LIN {X 0,Y 220.868,Z 520.969,A -85,B 0,C 180,E1 -20497.552,E2 -20497.552} C_VEL
LIN {X 0,Y 220.987,Z 520.957,A -85,B 0,C 180,E1 -20502.57,E2 -20502.57} C_VEL
LIN {X 0,Y 221.013,Z 520.952,A -85,B 0,C 180,E1 -20507.138,E2 -20507.138} C_VEL
LIN {X 0,Y 221.2,Z 520.932,A -85,B 0,C 180,E1 -20510.859,E2 -20510.859} C_VEL
LIN {X 0,Y 221.129,Z 520.939,A -85,B 0,C 180,E1 -20514.528,E2 -20514.528} C_VEL
LIN {X 0,Y 221.511,Z 520.89,A -85,B 0,C 180,E1 -20518.181,E2 -20518.181} C_VEL
LIN {X 0,Y 221.506,Z 520.891,A -85,B 0,C 180,E1 -20521.818,E2 -20521.818} C_VEL
LIN {X 0,Y 221.24,Z 520.926,A -85,B 0,C 180,E1 -20527.3,E2 -20527.3} C_VEL
LIN {X 0,Y 221.067,Z 520.947,A -85,B 0,C 180,E1 -20530.996,E2 -20530.996} C_VEL
LIN {X 0,Y 220.978,Z 520.958,A -85,B 0,C 180,E1 -20534.74,E2 -20534.74} C_VEL
LIN {X 0,Y 220.899,Z 520.969,A -85,B 0,C 180,E1 -20538.551,E2 -20538.551} C_VEL
LIN {X 0,Y 220.868,Z 520.97,A -85,B 0,C 180,E1 -20542.664,E2 -20542.664} C_VEL
LIN {X 0,Y 220.866,Z 520.973,A -85,B 0,C 180,E1 -20547.005,E2 -20547.005} C_VEL
LIN {X 0,Y 220.818,Z 520.98,A -85,B 0,C 180,E1 -20550.758,E2 -20550.758} C_VEL
LIN {X 0,Y 220.81,Z 520.981,A -85,B 0,C 180,E1 -20554.953,E2 -20554.953} C_VEL
LIN {X 0,Y 220.892,Z 521.149,A -85,B 0,C 180,E1 -20556.482,E2 -20556.482} C_VEL
LIN {X 0,Y 222.343,Z 528.666,A -85,B 0,C 180,E1 -20561.589,E2 -20561.589} C_VEL
LIN {X 0,Y 223.777,Z 535.991,A -85,B 0,C 180,E1 -20566.296,E2 -20566.296} C_VEL
LIN {X 0,Y 225.008,Z 542.365,A -85,B 0,C 180,E1 -20570.186,E2 -20570.186} C_VEL
LIN {X 0,Y 225.036,Z 544.358,A -85,B 0,C 180,E1 -20571.346,E2 -20571.346} C_VEL
LIN {X 0,Y 222.99,Z 553.544,A -85,B 0,C 180,E1 -20576.527,E2 -20576.527} C_VEL
LIN {X 0,Y 221.333,Z 562.382,A -85,B 0,C 180,E1 -20581.395,E2 -20581.395} C_VEL
LIN {X 0,Y 222.533,Z 577.013,A -85,B 0,C 180,E1 -20582.449,E2 -20582.449} C_VEL
LIN {X 0,Y 223.287,Z 589.6,A -85,B 0,C 180,E1 -20583.692,E2 -20583.692} C_VEL
LIN {X 0,Y 223.376,Z 591.056,A -85,B 0,C 180,E1 -20583.862,E2 -20583.862} C_VEL
LIN {X 0,Y 222.993,Z 596.491,A -85,B 0,C 180,E1 -20584.484,E2 -20584.484} C_VEL
LIN {X 0,Y 220.374,Z 605.07,A -85,B 0,C 180,E1 -20585.546,E2 -20585.546} C_VEL
LIN {X 0,Y 217.508,Z 613.354,A -85,B 0,C 180,E1 -20586.792,E2 -20586.792} C_VEL
LIN {X 0,Y 216.761,Z 618.17,A -85,B 0,C 180,E1 -20587.69,E2 -20587.69} C_VEL
LIN {X 0,Y 216.495,Z 628.791,A -85,B 0,C 180,E1 -20590.028,E2 -20590.028} C_VEL
LIN {X 0,Y 215.182,Z 637.685,A -85,B 0,C 180,E1 -20592.416,E2 -20592.416} C_VEL
LIN {X 0,Y 213.795,Z 646.126,A -85,B 0,C 180,E1 -20595.241,E2 -20595.241} C_VEL
LIN {X 0,Y 213.228,Z 652.944,A -85,B 0,C 180,E1 -20598.112,E2 -20598.112} C_VEL
LIN {X 0,Y 213.044,Z 659.023,A -85,B 0,C 180,E1 -20601.395,E2 -20601.395} C_VEL
LIN {X 0,Y 213.394,Z 663.111,A -85,B 0,C 180,E1 -20604.33,E2 -20604.33} C_VEL
LIN {X 0,Y 213.6,Z 665.077,A -85,B 0,C 180,E1 -20606.227,E2 -20606.227} C_VEL
LIN {X 0,Y 213.964,Z 666.582,A -85,B 0,C 180,E1 -20608.118,E2 -20608.118} C_VEL
LIN {X 0,Y 214.253,Z 667.619,A -85,B 0,C 180,E1 -20610,E2 -20610} C_VEL
LIN {X 0,Y 213.722,Z 668.07,A -85,B 0,C 180,E1 -20611.885,E2 -20611.885} C_VEL
LIN {X 0,Y 213.262,Z 668.071,A -85,B 0,C 180,E1 -20613.779,E2 -20613.779} C_VEL
LIN {X 0,Y 212.95,Z 667.676,A -85,B 0,C 180,E1 -20615.682,E2 -20615.682} C_VEL
LIN {X 0,Y 212.44,Z 665.683,A -85,B 0,C 180,E1 -20619.521,E2 -20619.521} C_VEL
LIN {X 0,Y 212.569,Z 664.115,A -85,B 0,C 180,E1 -20621.442,E2 -20621.442} C_VEL
LIN {X 0,Y 213.6,Z 659.748,A -85,B 0,C 180,E1 -20625.262,E2 -20625.262} C_VEL
LIN {X 0,Y 214.967,Z 655.403,A -85,B 0,C 180,E1 -20628.095,E2 -20628.095} C_VEL
LIN {X 0,Y 217.648,Z 649.066,A -85,B 0,C 180,E1 -20631.302,E2 -20631.302} C_VEL
LIN {X 0,Y 221.044,Z 641.112,A -85,B 0,C 180,E1 -20634.415,E2 -20634.415} C_VEL
LIN {X 0,Y 224.313,Z 631.288,A -85,B 0,C 180,E1 -20637.525,E2 -20637.525} C_VEL
LIN {X 0,Y 227.265,Z 621.289,A -85,B 0,C 180,E1 -20640.116,E2 -20640.116} C_VEL
LIN {X 0,Y 229.051,Z 612.146,A -85,B 0,C 180,E1 -20642.217,E2 -20642.217} C_VEL
LIN {X 0,Y 230.395,Z 601.122,A -85,B 0,C 180,E1 -20644.552,E2 -20644.552} C_VEL
LIN {X 0,Y 230.791,Z 590.585,A -85,B 0,C 180,E1 -20646.665,E2 -20646.665} C_VEL
LIN {X 0,Y 230.404,Z 579.42,A -85,B 0,C 180,E1 -20648.907,E2 -20648.907} C_VEL
LIN {X 0,Y 229.373,Z 570.02,A -85,B 0,C 180,E1 -20650.835,E2 -20650.835} C_VEL
LIN {X 0,Y 228.281,Z 563.015,A -85,B 0,C 180,E1 -20652.364,E2 -20652.364} C_VEL
LIN {X 0,Y 225.952,Z 556.827,A -85,B 0,C 180,E1 -20654.258,E2 -20654.258} C_VEL
LIN {X 0,Y 223.212,Z 551.163,A -85,B 0,C 180,E1 -20656.437,E2 -20656.437} C_VEL
LIN {X 0,Y 222.42,Z 548.881,A -85,B 0,C 180,E1 -20657.206,E2 -20657.206} C_VEL
LIN {X 0,Y 218.789,Z 542.503,A -85,B 0,C 180,E1 -20660.551,E2 -20660.551} C_VEL
LIN {X 0,Y 217.55,Z 538.888,A -85,B 0,C 180,E1 -20662.279,E2 -20662.279} C_VEL
LIN {X 0,Y 217.174,Z 536.934,A -85,B 0,C 180,E1 -20664.374,E2 -20664.374} C_VEL
LIN {X 0,Y 216.367,Z 533.433,A -85,B 0,C 180,E1 -20668.688,E2 -20668.688} C_VEL
LIN {X 0,Y 215.819,Z 530.571,A -85,B 0,C 180,E1 -20672.878,E2 -20672.878} C_VEL
LIN {X 0,Y 215.351,Z 528.348,A -85,B 0,C 180,E1 -20676.945,E2 -20676.945} C_VEL
LIN {X 0,Y 215.107,Z 527.422,A -85,B 0,C 180,E1 -20679.213,E2 -20679.213} C_VEL
LIN {X 0,Y 216.79,Z 529.004,A -85,B 0,C 180,E1 -20682.175,E2 -20682.175} C_VEL
LIN {X 0,Y 219.429,Z 530.078,A -85,B 0,C 180,E1 -20685.154,E2 -20685.154} C_VEL
LIN {X 0,Y 220.989,Z 532.089,A -85,B 0,C 180,E1 -20686.904,E2 -20686.904} C_VEL
LIN {X 0,Y 222.543,Z 533.032,A -85,B 0,C 180,E1 -20688.238,E2 -20688.238} C_VEL
LIN {X 0,Y 224.34,Z 536.433,A -85,B 0,C 180,E1 -20690.145,E2 -20690.145} C_VEL
LIN {X 0,Y 225.36,Z 537.698,A -85,B 0,C 180,E1 -20691.03,E2 -20691.03} C_VEL
LIN {X 0,Y 230.369,Z 546.87,A -85,B 0,C 180,E1 -20695.625,E2 -20695.625} C_VEL
LIN {X 0,Y 232.402,Z 551.236,A -85,B 0,C 180,E1 -20697.547,E2 -20697.547} C_VEL
LIN {X 0,Y 235.12,Z 559.958,A -85,B 0,C 180,E1 -20700.857,E2 -20700.857} C_VEL
LIN {X 0,Y 236.611,Z 566.893,A -85,B 0,C 180,E1 -20703.406,E2 -20703.406} C_VEL
LIN {X 0,Y 237.291,Z 573.898,A -85,B 0,C 180,E1 -20705.951,E2 -20705.951} C_VEL
LIN {X 0,Y 233.871,Z 582.058,A -85,B 0,C 180,E1 -20708.135,E2 -20708.135} C_VEL
LIN {X 0,Y 230.347,Z 589.283,A -85,B 0,C 180,E1 -20710.549,E2 -20710.549} C_VEL
LIN {X 0,Y 226.712,Z 595.941,A -85,B 0,C 180,E1 -20713.445,E2 -20713.445} C_VEL
LIN {X 0,Y 223.496,Z 601.099,A -85,B 0,C 180,E1 -20716.441,E2 -20716.441} C_VEL
LIN {X 0,Y 220.741,Z 604.875,A -85,B 0,C 180,E1 -20719.531,E2 -20719.531} C_VEL
LIN {X 0,Y 218.492,Z 607.379,A -85,B 0,C 180,E1 -20722.706,E2 -20722.706} C_VEL
LIN {X 0,Y 217.166,Z 608.443,A -85,B 0,C 180,E1 -20725.021,E2 -20725.021} C_VEL
LIN {X 0,Y 215.688,Z 608.843,A -85,B 0,C 180,E1 -20728.384,E2 -20728.384} C_VEL
LIN {X 0,Y 214.787,Z 608.01,A -85,B 0,C 180,E1 -20731.707,E2 -20731.707} C_VEL
LIN {X 0,Y 214.36,Z 606.025,A -85,B 0,C 180,E1 -20734.95,E2 -20734.95} C_VEL
LIN {X 0,Y 214.38,Z 602.431,A -85,B 0,C 180,E1 -20738.527,E2 -20738.527} C_VEL
LIN {X 0,Y 214.977,Z 597.143,A -85,B 0,C 180,E1 -20742.145,E2 -20742.145} C_VEL
LIN {X 0,Y 215.807,Z 591.954,A -85,B 0,C 180,E1 -20744.852,E2 -20744.852} C_VEL
LIN {X 0,Y 216.835,Z 585.672,A -85,B 0,C 180,E1 -20747.512,E2 -20747.512} C_VEL
LIN {X 0,Y 218.123,Z 578.071,A -85,B 0,C 180,E1 -20750.135,E2 -20750.135} C_VEL
LIN {X 0,Y 219.642,Z 569.436,A -85,B 0,C 180,E1 -20752.558,E2 -20752.558} C_VEL
LIN {X 0,Y 221.381,Z 558.618,A -85,B 0,C 180,E1 -20755.028,E2 -20755.028} C_VEL
LIN {X 0,Y 222.361,Z 551.653,A -85,B 0,C 180,E1 -20756.349,E2 -20756.349} C_VEL
LIN {X 0,Y 219.673,Z 541.039,A -85,B 0,C 180,E1 -20758.406,E2 -20758.406} C_VEL
LIN {X 0,Y 216.303,Z 529.758,A -85,B 0,C 180,E1 -20760.297,E2 -20760.297} C_VEL
LIN {X 0,Y 213.826,Z 521.856,A -85,B 0,C 180,E1 -20761.471,E2 -20761.471} C_VEL
LIN {X 0,Y 213.803,Z 521.854,A -85,B 0,C 180,E1 -20764.701,E2 -20764.701} C_VEL
LIN {X 0,Y 213.802,Z 521.852,A -85,B 0,C 180,E1 -20768.802,E2 -20768.802} C_VEL
LIN {X 0,Y 213.926,Z 521.838,A -85,B 0,C 180,E1 -20772.802,E2 -20772.802} C_VEL
LIN {X 0,Y 213.948,Z 521.835,A -85,B 0,C 180,E1 -20776.706,E2 -20776.706} C_VEL
LIN {X 0,Y 214.14,Z 521.81,A -85,B 0,C 180,E1 -20780.555,E2 -20780.555} C_VEL
LIN {X 0,Y 214.093,Z 521.815,A -85,B 0,C 180,E1 -20784.348,E2 -20784.348} C_VEL
LIN {X 0,Y 214.447,Z 521.77,A -85,B 0,C 180,E1 -20788.122,E2 -20788.122} C_VEL
LIN {X 0,Y 214.54,Z 521.759,A -85,B 0,C 180,E1 -20790,E2 -20790} C_VEL
LIN {X 0,Y 214.446,Z 521.771,A -85,B 0,C 180,E1 -20791.878,E2 -20791.878} C_VEL
LIN {X 0,Y 214.185,Z 521.802,A -85,B 0,C 180,E1 -20797.542,E2 -20797.542} C_VEL
LIN {X 0,Y 213.998,Z 521.83,A -85,B 0,C 180,E1 -20801.364,E2 -20801.364} C_VEL
LIN {X 0,Y 213.921,Z 521.838,A -85,B 0,C 180,E1 -20805.238,E2 -20805.238} C_VEL
LIN {X 0,Y 213.838,Z 521.848,A -85,B 0,C 180,E1 -20809.187,E2 -20809.187} C_VEL
LIN {X 0,Y 213.808,Z 521.852,A -85,B 0,C 180,E1 -20813.231,E2 -20813.231} C_VEL
LIN {X 0,Y 213.792,Z 521.854,A -85,B 0,C 180,E1 -20817.428,E2 -20817.428} C_VEL
LIN {X 0,Y 213.761,Z 521.856,A -85,B 0,C 180,E1 -20821.738,E2 -20821.738} C_VEL
LIN {X 0,Y 213.746,Z 521.857,A -85,B 0,C 180,E1 -20826.288,E2 -20826.288} C_VEL
LIN {X 0,Y 213.705,Z 521.864,A -85,B 0,C 180,E1 -20831.127,E2 -20831.127} C_VEL
LIN {X 0,Y 213.705,Z 521.862,A -85,B 0,C 180,E1 -20833.679,E2 -20833.679} C_VEL
LIN {X 0,Y 213.705,Z 521.863,A -85,B 0,C 180,E1 -20836.344,E2 -20836.344} C_VEL
LIN {X 0,Y 213.719,Z 521.863,A -85,B 0,C 180,E1 -20839.143,E2 -20839.143} C_VEL
LIN {X 0,Y 213.746,Z 521.858,A -85,B 0,C 180,E1 -20843.711,E2 -20843.711} C_VEL
LIN {X 0,Y 213.797,Z 521.852,A -85,B 0,C 180,E1 -20848.724,E2 -20848.724} C_VEL
LIN {X 0,Y 213.828,Z 521.848,A -85,B 0,C 180,E1 -20852.603,E2 -20852.603} C_VEL
LIN {X 0,Y 213.821,Z 521.85,A -85,B 0,C 180,E1 -20856.973,E2 -20856.973} C_VEL
LIN {X 0,Y 213.946,Z 521.836,A -85,B 0,C 180,E1 -20862.803,E2 -20862.803} C_VEL
LIN {X 0,Y 213.955,Z 521.832,A -85,B 0,C 180,E1 -20866.706,E2 -20866.706} C_VEL
LIN {X 0,Y 214.138,Z 521.81,A -85,B 0,C 180,E1 -20870.555,E2 -20870.555} C_VEL
LIN {X 0,Y 214.09,Z 521.815,A -85,B 0,C 180,E1 -20874.348,E2 -20874.348} C_VEL
LIN {X 0,Y 214.444,Z 521.77,A -85,B 0,C 180,E1 -20878.121,E2 -20878.121} C_VEL
LIN {X 0,Y 214.543,Z 521.759,A -85,B 0,C 180,E1 -20880,E2 -20880} C_VEL
LIN {X 0,Y 214.439,Z 521.771,A -85,B 0,C 180,E1 -20881.878,E2 -20881.878} C_VEL
LIN {X 0,Y 214.182,Z 521.804,A -85,B 0,C 180,E1 -20887.542,E2 -20887.542} C_VEL
LIN {X 0,Y 213.998,Z 521.825,A -85,B 0,C 180,E1 -20891.364,E2 -20891.364} C_VEL
LIN {X 0,Y 213.914,Z 521.838,A -85,B 0,C 180,E1 -20895.238,E2 -20895.238} C_VEL
LIN {X 0,Y 213.82,Z 521.849,A -85,B 0,C 180,E1 -20899.189,E2 -20899.189} C_VEL
LIN {X 0,Y 213.803,Z 521.851,A -85,B 0,C 180,E1 -20903.232,E2 -20903.232} C_VEL
LIN {X 0,Y 213.787,Z 521.853,A -85,B 0,C 180,E1 -20907.428,E2 -20907.428} C_VEL
LIN {X 0,Y 213.759,Z 521.861,A -85,B 0,C 180,E1 -20911.739,E2 -20911.739} C_VEL
LIN {X 0,Y 213.83,Z 522.009,A -85,B 0,C 180,E1 -20916.053,E2 -20916.053} C_VEL
LIN {X 0,Y 215.117,Z 528.734,A -85,B 0,C 180,E1 -20920.799,E2 -20920.799} C_VEL
LIN {X 0,Y 216.124,Z 533.968,A -85,B 0,C 180,E1 -20924.324,E2 -20924.324} C_VEL
LIN {X 0,Y 217.586,Z 541.147,A -85,B 0,C 180,E1 -20928.934,E2 -20928.934} C_VEL
LIN {X 0,Y 217.963,Z 544.027,A -85,B 0,C 180,E1 -20930.701,E2 -20930.701} C_VEL
LIN {X 0,Y 217.58,Z 546.471,A -85,B 0,C 180,E1 -20932.141,E2 -20932.141} C_VEL
LIN {X 0,Y 215.903,Z 553.764,A -85,B 0,C 180,E1 -20936.401,E2 -20936.401} C_VEL
LIN {X 0,Y 214.425,Z 561.289,A -85,B 0,C 180,E1 -20940.752,E2 -20940.752} C_VEL
LIN {X 0,Y 215.6,Z 576.166,A -85,B 0,C 180,E1 -20941.87,E2 -20941.87} C_VEL
LIN {X 0,Y 216.289,Z 589.084,A -85,B 0,C 180,E1 -20943.202,E2 -20943.202} C_VEL
LIN {X 0,Y 216.665,Z 601.267,A -85,B 0,C 180,E1 -20944.803,E2 -20944.803} C_VEL
LIN {X 0,Y 216.83,Z 612.403,A -85,B 0,C 180,E1 -20946.606,E2 -20946.606} C_VEL
LIN {X 0,Y 216.761,Z 618.17,A -85,B 0,C 180,E1 -20947.69,E2 -20947.69} C_VEL
LIN {X 0,Y 215.93,Z 622.846,A -85,B 0,C 180,E1 -20948.642,E2 -20948.642} C_VEL
LIN {X 0,Y 214.068,Z 627.214,A -85,B 0,C 180,E1 -20949.61,E2 -20949.61} C_VEL
LIN {X 0,Y 209.48,Z 635.189,A -85,B 0,C 180,E1 -20951.703,E2 -20951.703} C_VEL
LIN {X 0,Y 207.845,Z 638.989,A -85,B 0,C 180,E1 -20952.892,E2 -20952.892} C_VEL
LIN {X 0,Y 207.543,Z 640.232,A -85,B 0,C 180,E1 -20953.312,E2 -20953.312} C_VEL
LIN {X 0,Y 206.563,Z 647.939,A -85,B 0,C 180,E1 -20956.222,E2 -20956.222} C_VEL
LIN {X 0,Y 206.06,Z 654.149,A -85,B 0,C 180,E1 -20959.188,E2 -20959.188} C_VEL
LIN {X 0,Y 206.046,Z 659.04,A -85,B 0,C 180,E1 -20962.159,E2 -20962.159} C_VEL
LIN {X 0,Y 206.462,Z 662.744,A -85,B 0,C 180,E1 -20965.118,E2 -20965.118} C_VEL
LIN {X 0,Y 206.931,Z 665.294,A -85,B 0,C 180,E1 -20968.054,E2 -20968.054} C_VEL
LIN {X 0,Y 207.253,Z 666.387,A -85,B 0,C 180,E1 -20970,E2 -20970} C_VEL
LIN {X 0,Y 206.697,Z 666.887,A -85,B 0,C 180,E1 -20971.949,E2 -20971.949} C_VEL
LIN {X 0,Y 206.201,Z 666.971,A -85,B 0,C 180,E1 -20973.909,E2 -20973.909} C_VEL
LIN {X 0,Y 205.879,Z 666.632,A -85,B 0,C 180,E1 -20975.878,E2 -20975.878} C_VEL
LIN {X 0,Y 205.38,Z 664.743,A -85,B 0,C 180,E1 -20979.852,E2 -20979.852} C_VEL
LIN {X 0,Y 205.954,Z 661.373,A -85,B 0,C 180,E1 -20983.82,E2 -20983.82} C_VEL
LIN {X 0,Y 207.628,Z 656.377,A -85,B 0,C 180,E1 -20987.737,E2 -20987.737} C_VEL
LIN {X 0,Y 209.681,Z 651.515,A -85,B 0,C 180,E1 -20990.606,E2 -20990.606} C_VEL
LIN {X 0,Y 212.984,Z 644.514,A -85,B 0,C 180,E1 -20993.843,E2 -20993.843} C_VEL
LIN {X 0,Y 215.983,Z 637.184,A -85,B 0,C 180,E1 -20996.579,E2 -20996.579} C_VEL
LIN {X 0,Y 219.013,Z 628.599,A -85,B 0,C 180,E1 -20999.234,E2 -20999.234} C_VEL
LIN {X 0,Y 222.103,Z 617.956,A -85,B 0,C 180,E1 -21002.007,E2 -21002.007} C_VEL
LIN {X 0,Y 224.097,Z 606.805,A -85,B 0,C 180,E1 -21004.631,E2 -21004.631} C_VEL
LIN {X 0,Y 225.205,Z 596.058,A -85,B 0,C 180,E1 -21006.971,E2 -21006.971} C_VEL
LIN {X 0,Y 225.365,Z 583.627,A -85,B 0,C 180,E1 -21009.637,E2 -21009.637} C_VEL
LIN {X 0,Y 224.586,Z 571.366,A -85,B 0,C 180,E1 -21012.343,E2 -21012.343} C_VEL
LIN {X 0,Y 224.02,Z 567.653,A -85,B 0,C 180,E1 -21013.235,E2 -21013.235} C_VEL
LIN {X 0,Y 222.549,Z 562.746,A -85,B 0,C 180,E1 -21014.783,E2 -21014.783} C_VEL
LIN {X 0,Y 219.891,Z 556.62,A -85,B 0,C 180,E1 -21017.241,E2 -21017.241} C_VEL
LIN {X 0,Y 219.193,Z 554.511,A -85,B 0,C 180,E1 -21018.048,E2 -21018.048} C_VEL
LIN {X 0,Y 215.995,Z 547.879,A -85,B 0,C 180,E1 -21021.591,E2 -21021.591} C_VEL
LIN {X 0,Y 215.084,Z 545.09,A -85,B 0,C 180,E1 -21022.995,E2 -21022.995} C_VEL
LIN {X 0,Y 212.196,Z 539.413,A -85,B 0,C 180,E1 -21028.419,E2 -21028.419} C_VEL
LIN {X 0,Y 211.575,Z 536.634,A -85,B 0,C 180,E1 -21032.287,E2 -21032.287} C_VEL
LIN {X 0,Y 212.378,Z 534.76,A -85,B 0,C 180,E1 -21037.119,E2 -21037.119} C_VEL
LIN {X 0,Y 213.373,Z 534.411,A -85,B 0,C 180,E1 -21039.263,E2 -21039.263} C_VEL
LIN {X 0,Y 215.359,Z 536.111,A -85,B 0,C 180,E1 -21042.921,E2 -21042.921} C_VEL
LIN {X 0,Y 217.092,Z 536.896,A -85,B 0,C 180,E1 -21044.99,E2 -21044.99} C_VEL
LIN {X 0,Y 218.737,Z 538.899,A -85,B 0,C 180,E1 -21047.003,E2 -21047.003} C_VEL
LIN {X 0,Y 219.815,Z 539.821,A -85,B 0,C 180,E1 -21048.09,E2 -21048.09} C_VEL
LIN {X 0,Y 222.545,Z 545.038,A -85,B 0,C 180,E1 -21051.307,E2 -21051.307} C_VEL
LIN {X 0,Y 226.246,Z 552.522,A -85,B 0,C 180,E1 -21055.301,E2 -21055.301} C_VEL
LIN {X 0,Y 227.969,Z 556.735,A -85,B 0,C 180,E1 -21057.254,E2 -21057.254} C_VEL
LIN {X 0,Y 230.367,Z 566.269,A -85,B 0,C 180,E1 -21061.131,E2 -21061.131} C_VEL
LIN {X 0,Y 231.268,Z 573.398,A -85,B 0,C 180,E1 -21063.921,E2 -21063.921} C_VEL
LIN {X 0,Y 231.367,Z 576.788,A -85,B 0,C 180,E1 -21065.229,E2 -21065.229} C_VEL
LIN {X 0,Y 227.544,Z 584.936,A -85,B 0,C 180,E1 -21067.557,E2 -21067.557} C_VEL
LIN {X 0,Y 223.344,Z 592.775,A -85,B 0,C 180,E1 -21070.425,E2 -21070.425} C_VEL
LIN {X 0,Y 220.216,Z 598.009,A -85,B 0,C 180,E1 -21072.909,E2 -21072.909} C_VEL
LIN {X 0,Y 216.841,Z 602.912,A -85,B 0,C 180,E1 -21075.992,E2 -21075.992} C_VEL
LIN {X 0,Y 213.967,Z 606.475,A -85,B 0,C 180,E1 -21079.176,E2 -21079.176} C_VEL
LIN {X 0,Y 211.991,Z 608.442,A -85,B 0,C 180,E1 -21081.833,E2 -21081.833} C_VEL
LIN {X 0,Y 209.967,Z 609.808,A -85,B 0,C 180,E1 -21085.344,E2 -21085.344} C_VEL
LIN {X 0,Y 208.5,Z 609.88,A -85,B 0,C 180,E1 -21088.789,E2 -21088.789} C_VEL
LIN {X 0,Y 207.648,Z 608.693,A -85,B 0,C 180,E1 -21092.204,E2 -21092.204} C_VEL
LIN {X 0,Y 207.279,Z 606.371,A -85,B 0,C 180,E1 -21095.536,E2 -21095.536} C_VEL
LIN {X 0,Y 207.353,Z 602.965,A -85,B 0,C 180,E1 -21098.779,E2 -21098.779} C_VEL
LIN {X 0,Y 207.858,Z 598.439,A -85,B 0,C 180,E1 -21101.939,E2 -21101.939} C_VEL
LIN {X 0,Y 208.787,Z 592.729,A -85,B 0,C 180,E1 -21105.017,E2 -21105.017} C_VEL
LIN {X 0,Y 209.913,Z 585.863,A -85,B 0,C 180,E1 -21107.962,E2 -21107.962} C_VEL
LIN {X 0,Y 211.369,Z 577.551,A -85,B 0,C 180,E1 -21110.82,E2 -21110.82} C_VEL
LIN {X 0,Y 213.189,Z 567.487,A -85,B 0,C 180,E1 -21113.602,E2 -21113.602} C_VEL
LIN {X 0,Y 214.866,Z 557.035,A -85,B 0,C 180,E1 -21115.911,E2 -21115.911} C_VEL
LIN {X 0,Y 215.445,Z 553.444,A -85,B 0,C 180,E1 -21116.6,E2 -21116.6} C_VEL
LIN {X 0,Y 213.299,Z 544.314,A -85,B 0,C 180,E1 -21118.461,E2 -21118.461} C_VEL
LIN {X 0,Y 209.808,Z 532.392,A -85,B 0,C 180,E1 -21120.593,E2 -21120.593} C_VEL
LIN {X 0,Y 206.77,Z 522.733,A -85,B 0,C 180,E1 -21122.097,E2 -21122.097} C_VEL
LIN {X 0,Y 206.758,Z 522.73,A -85,B 0,C 180,E1 -21126.604,E2 -21126.604} C_VEL
LIN {X 0,Y 206.872,Z 522.716,A -85,B 0,C 180,E1 -21132.196,E2 -21132.196} C_VEL
LIN {X 0,Y 206.889,Z 522.714,A -85,B 0,C 180,E1 -21136.244,E2 -21136.244} C_VEL
LIN {X 0,Y 207.084,Z 522.689,A -85,B 0,C 180,E1 -21140.23,E2 -21140.23} C_VEL
LIN {X 0,Y 207.055,Z 522.692,A -85,B 0,C 180,E1 -21144.155,E2 -21144.155} C_VEL
LIN {X 0,Y 207.384,Z 522.65,A -85,B 0,C 180,E1 -21148.058,E2 -21148.058} C_VEL
LIN {X 0,Y 207.507,Z 522.636,A -85,B 0,C 180,E1 -21150,E2 -21150} C_VEL
LIN {X 0,Y 207.382,Z 522.65,A -85,B 0,C 180,E1 -21151.942,E2 -21151.942} C_VEL
LIN {X 0,Y 207.13,Z 522.68,A -85,B 0,C 180,E1 -21157.8,E2 -21157.8} C_VEL
LIN {X 0,Y 206.921,Z 522.709,A -85,B 0,C 180,E1 -21161.758,E2 -21161.758} C_VEL
LIN {X 0,Y 206.857,Z 522.715,A -85,B 0,C 180,E1 -21165.771,E2 -21165.771} C_VEL
LIN {X 0,Y 206.766,Z 522.727,A -85,B 0,C 180,E1 -21169.871,E2 -21169.871} C_VEL
LIN {X 0,Y 206.743,Z 522.729,A -85,B 0,C 180,E1 -21174.074,E2 -21174.074} C_VEL
LIN {X 0,Y 206.693,Z 522.736,A -85,B 0,C 180,E1 -21178.426,E2 -21178.426} C_VEL
LIN {X 0,Y 206.698,Z 522.738,A -85,B 0,C 180,E1 -21182.958,E2 -21182.958} C_VEL
LIN {X 0,Y 206.676,Z 522.739,A -85,B 0,C 180,E1 -21187.741,E2 -21187.741} C_VEL
LIN {X 0,Y 206.637,Z 522.742,A -85,B 0,C 180,E1 -21191.56,E2 -21191.56} C_VEL
LIN {X 0,Y 206.633,Z 522.745,A -85,B 0,C 180,E1 -21195.582,E2 -21195.582} C_VEL
LIN {X 0,Y 206.662,Z 522.739,A -85,B 0,C 180,E1 -21199.748,E2 -21199.748} C_VEL
LIN {X 0,Y 206.701,Z 522.736,A -85,B 0,C 180,E1 -21204.688,E2 -21204.688} C_VEL
LIN {X 0,Y 206.725,Z 522.73,A -85,B 0,C 180,E1 -21209.339,E2 -21209.339} C_VEL
LIN {X 0,Y 206.733,Z 522.732,A -85,B 0,C 180,E1 -21213.771,E2 -21213.771} C_VEL
LIN {X 0,Y 206.741,Z 522.728,A -85,B 0,C 180,E1 -21218.041,E2 -21218.041} C_VEL
LIN {X 0,Y 206.875,Z 522.714,A -85,B 0,C 180,E1 -21222.196,E2 -21222.196} C_VEL
LIN {X 0,Y 206.898,Z 522.709,A -85,B 0,C 180,E1 -21226.244,E2 -21226.244} C_VEL
LIN {X 0,Y 207.081,Z 522.688,A -85,B 0,C 180,E1 -21230.23,E2 -21230.23} C_VEL
LIN {X 0,Y 207.052,Z 522.691,A -85,B 0,C 180,E1 -21234.155,E2 -21234.155} C_VEL
LIN {X 0,Y 207.38,Z 522.65,A -85,B 0,C 180,E1 -21238.057,E2 -21238.057} C_VEL
LIN {X 0,Y 207.509,Z 522.635,A -85,B 0,C 180,E1 -21239.999,E2 -21239.999} C_VEL
LIN {X 0,Y 207.375,Z 522.651,A -85,B 0,C 180,E1 -21241.942,E2 -21241.942} C_VEL
LIN {X 0,Y 207.127,Z 522.682,A -85,B 0,C 180,E1 -21247.8,E2 -21247.8} C_VEL
LIN {X 0,Y 206.922,Z 522.706,A -85,B 0,C 180,E1 -21251.758,E2 -21251.758} C_VEL
LIN {X 0,Y 206.847,Z 522.717,A -85,B 0,C 180,E1 -21255.772,E2 -21255.772} C_VEL
LIN {X 0,Y 206.857,Z 522.716,A -85,B 0,C 180,E1 -21257.954,E2 -21257.954} C_VEL
LIN {X 0,Y 206.746,Z 522.73,A -85,B 0,C 180,E1 -21263.39,E2 -21263.39} C_VEL
LIN {X 0,Y 206.689,Z 522.738,A -85,B 0,C 180,E1 -21268.427,E2 -21268.427} C_VEL
LIN {X 0,Y 206.697,Z 522.741,A -85,B 0,C 180,E1 -21272.958,E2 -21272.958} C_VEL
LIN {X 0,Y 206.778,Z 522.885,A -85,B 0,C 180,E1 -21275.646,E2 -21275.646} C_VEL
LIN {X 0,Y 207.894,Z 528.772,A -85,B 0,C 180,E1 -21279.964,E2 -21279.964} C_VEL
LIN {X 0,Y 208.919,Z 533.975,A -85,B 0,C 180,E1 -21283.599,E2 -21283.599} C_VEL
LIN {X 0,Y 210.272,Z 540.642,A -85,B 0,C 180,E1 -21288.051,E2 -21288.051} C_VEL
LIN {X 0,Y 210.883,Z 544.806,A -85,B 0,C 180,E1 -21290.713,E2 -21290.713} C_VEL
LIN {X 0,Y 209.874,Z 549.36,A -85,B 0,C 180,E1 -21293.483,E2 -21293.483} C_VEL
LIN {X 0,Y 208.365,Z 555.987,A -85,B 0,C 180,E1 -21297.482,E2 -21297.482} C_VEL
LIN {X 0,Y 207.508,Z 560.273,A -85,B 0,C 180,E1 -21300.065,E2 -21300.065} C_VEL
LIN {X 0,Y 208.674,Z 575.929,A -85,B 0,C 180,E1 -21301.304,E2 -21301.304} C_VEL
LIN {X 0,Y 209.337,Z 589.369,A -85,B 0,C 180,E1 -21302.779,E2 -21302.779} C_VEL
LIN {X 0,Y 209.668,Z 601.548,A -85,B 0,C 180,E1 -21304.473,E2 -21304.473} C_VEL
LIN {X 0,Y 209.784,Z 613.555,A -85,B 0,C 180,E1 -21306.558,E2 -21306.558} C_VEL
LIN {X 0,Y 209.567,Z 624.575,A -85,B 0,C 180,E1 -21308.907,E2 -21308.907} C_VEL
LIN {X 0,Y 209.255,Z 630.454,A -85,B 0,C 180,E1 -21310.375,E2 -21310.375} C_VEL
LIN {X 0,Y 207.847,Z 638.667,A -85,B 0,C 180,E1 -21312.791,E2 -21312.791} C_VEL
LIN {X 0,Y 207.543,Z 640.232,A -85,B 0,C 180,E1 -21313.312,E2 -21313.312} C_VEL
LIN {X 0,Y 206.299,Z 643.767,A -85,B 0,C 180,E1 -21314.585,E2 -21314.585} C_VEL
LIN {X 0,Y 202.81,Z 648.792,A -85,B 0,C 180,E1 -21316.778,E2 -21316.778} C_VEL
LIN {X 0,Y 199.677,Z 653.18,A -85,B 0,C 180,E1 -21319.157,E2 -21319.157} C_VEL
LIN {X 0,Y 198.997,Z 655.644,A -85,B 0,C 180,E1 -21320.684,E2 -21320.684} C_VEL
LIN {X 0,Y 199.29,Z 660.154,A -85,B 0,C 180,E1 -21323.927,E2 -21323.927} C_VEL
LIN {X 0,Y 199.535,Z 662.306,A -85,B 0,C 180,E1 -21325.961,E2 -21325.961} C_VEL
LIN {X 0,Y 199.897,Z 663.978,A -85,B 0,C 180,E1 -21327.985,E2 -21327.985} C_VEL
LIN {X 0,Y 200.248,Z 665.132,A -85,B 0,C 180,E1 -21330,E2 -21330} C_VEL
LIN {X 0,Y 199.667,Z 665.683,A -85,B 0,C 180,E1 -21332.017,E2 -21332.017} C_VEL
LIN {X 0,Y 198.787,Z 665.575,A -85,B 0,C 180,E1 -21336.089,E2 -21336.089} C_VEL
LIN {X 0,Y 198.347,Z 663.816,A -85,B 0,C 180,E1 -21340.205,E2 -21340.205} C_VEL
LIN {X 0,Y 199.001,Z 660.586,A -85,B 0,C 180,E1 -21344.313,E2 -21344.313} C_VEL
LIN {X 0,Y 200.247,Z 657.129,A -85,B 0,C 180,E1 -21347.357,E2 -21347.357} C_VEL
LIN {X 0,Y 202.138,Z 652.758,A -85,B 0,C 180,E1 -21350.346,E2 -21350.346} C_VEL
LIN {X 0,Y 205.4,Z 646.414,A -85,B 0,C 180,E1 -21353.706,E2 -21353.706} C_VEL
LIN {X 0,Y 208.592,Z 639.711,A -85,B 0,C 180,E1 -21356.515,E2 -21356.515} C_VEL
LIN {X 0,Y 212.302,Z 630.231,A -85,B 0,C 180,E1 -21359.773,E2 -21359.773} C_VEL
LIN {X 0,Y 215.602,Z 620.479,A -85,B 0,C 180,E1 -21362.538,E2 -21362.538} C_VEL
LIN {X 0,Y 218.153,Z 609.035,A -85,B 0,C 180,E1 -21365.443,E2 -21365.443} C_VEL
LIN {X 0,Y 219.586,Z 598.979,A -85,B 0,C 180,E1 -21367.805,E2 -21367.805} C_VEL
LIN {X 0,Y 220.258,Z 586.55,A -85,B 0,C 180,E1 -21370.664,E2 -21370.664} C_VEL
LIN {X 0,Y 219.965,Z 574.854,A -85,B 0,C 180,E1 -21373.424,E2 -21373.424} C_VEL
LIN {X 0,Y 219.702,Z 572.149,A -85,B 0,C 180,E1 -21374.131,E2 -21374.131} C_VEL
LIN {X 0,Y 218.547,Z 567.755,A -85,B 0,C 180,E1 -21375.619,E2 -21375.619} C_VEL
LIN {X 0,Y 216.657,Z 562.868,A -85,B 0,C 180,E1 -21377.694,E2 -21377.694} C_VEL
LIN {X 0,Y 216.196,Z 561.03,A -85,B 0,C 180,E1 -21378.39,E2 -21378.39} C_VEL
LIN {X 0,Y 212.915,Z 552.728,A -85,B 0,C 180,E1 -21382.838,E2 -21382.838} C_VEL
LIN {X 0,Y 212.372,Z 551.113,A -85,B 0,C 180,E1 -21383.789,E2 -21383.789} C_VEL
LIN {X 0,Y 210.037,Z 545.834,A -85,B 0,C 180,E1 -21389.03,E2 -21389.03} C_VEL
LIN {X 0,Y 209.617,Z 543.083,A -85,B 0,C 180,E1 -21393.088,E2 -21393.088} C_VEL
LIN {X 0,Y 210.933,Z 541.266,A -85,B 0,C 180,E1 -21398.5,E2 -21398.5} C_VEL
LIN {X 0,Y 214.432,Z 543.481,A -85,B 0,C 180,E1 -21404.8,E2 -21404.8} C_VEL
LIN {X 0,Y 216.804,Z 546.392,A -85,B 0,C 180,E1 -21407.922,E2 -21407.922} C_VEL
LIN {X 0,Y 219.895,Z 553.112,A -85,B 0,C 180,E1 -21412.219,E2 -21412.219} C_VEL
LIN {X 0,Y 222.633,Z 559.609,A -85,B 0,C 180,E1 -21415.803,E2 -21415.803} C_VEL
LIN {X 0,Y 224.157,Z 565.951,A -85,B 0,C 180,E1 -21418.653,E2 -21418.653} C_VEL
LIN {X 0,Y 225.337,Z 573.186,A -85,B 0,C 180,E1 -21421.788,E2 -21421.788} C_VEL
LIN {X 0,Y 225.523,Z 579.059,A -85,B 0,C 180,E1 -21424.267,E2 -21424.267} C_VEL
LIN {X 0,Y 223.014,Z 584.536,A -85,B 0,C 180,E1 -21425.879,E2 -21425.879} C_VEL
LIN {X 0,Y 219.039,Z 591.716,A -85,B 0,C 180,E1 -21428.381,E2 -21428.381} C_VEL
LIN {X 0,Y 215.018,Z 598.154,A -85,B 0,C 180,E1 -21431.31,E2 -21431.31} C_VEL
LIN {X 0,Y 211.649,Z 602.847,A -85,B 0,C 180,E1 -21434.124,E2 -21434.124} C_VEL
LIN {X 0,Y 208.116,Z 607.115,A -85,B 0,C 180,E1 -21437.694,E2 -21437.694} C_VEL
LIN {X 0,Y 206.284,Z 608.923,A -85,B 0,C 180,E1 -21439.92,E2 -21439.92} C_VEL
LIN {X 0,Y 204.711,Z 610.197,A -85,B 0,C 180,E1 -21442.189,E2 -21442.189} C_VEL
LIN {X 0,Y 202.757,Z 611.081,A -85,B 0,C 180,E1 -21445.681,E2 -21445.681} C_VEL
LIN {X 0,Y 201.323,Z 610.756,A -85,B 0,C 180,E1 -21449.258,E2 -21449.258} C_VEL
LIN {X 0,Y 200.519,Z 609.256,A -85,B 0,C 180,E1 -21452.735,E2 -21452.735} C_VEL
LIN {X 0,Y 200.2,Z 606.154,A -85,B 0,C 180,E1 -21456.641,E2 -21456.641} C_VEL
LIN {X 0,Y 200.507,Z 601.505,A -85,B 0,C 180,E1 -21460.513,E2 -21460.513} C_VEL
LIN {X 0,Y 201.411,Z 595.304,A -85,B 0,C 180,E1 -21464.258,E2 -21464.258} C_VEL
LIN {X 0,Y 202.534,Z 588.675,A -85,B 0,C 180,E1 -21467.365,E2 -21467.365} C_VEL
LIN {X 0,Y 203.8,Z 581.442,A -85,B 0,C 180,E1 -21470.112,E2 -21470.112} C_VEL
LIN {X 0,Y 205.613,Z 571.879,A -85,B 0,C 180,E1 -21473.034,E2 -21473.034} C_VEL
LIN {X 0,Y 207.496,Z 560.945,A -85,B 0,C 180,E1 -21475.702,E2 -21475.702} C_VEL
LIN {X 0,Y 208.544,Z 554.152,A -85,B 0,C 180,E1 -21477.083,E2 -21477.083} C_VEL
LIN {X 0,Y 205.643,Z 543.028,A -85,B 0,C 180,E1 -21479.423,E2 -21479.423} C_VEL
LIN {X 0,Y 202.695,Z 532.887,A -85,B 0,C 180,E1 -21481.258,E2 -21481.258} C_VEL
LIN {X 0,Y 199.7,Z 523.613,A -85,B 0,C 180,E1 -21482.773,E2 -21482.773} C_VEL
LIN {X 0,Y 199.717,Z 523.608,A -85,B 0,C 180,E1 -21487.226,E2 -21487.226} C_VEL
LIN {X 0,Y 199.799,Z 523.598,A -85,B 0,C 180,E1 -21491.759,E2 -21491.759} C_VEL
LIN {X 0,Y 199.828,Z 523.595,A -85,B 0,C 180,E1 -21495.747,E2 -21495.747} C_VEL
LIN {X 0,Y 200.027,Z 523.569,A -85,B 0,C 180,E1 -21499.882,E2 -21499.882} C_VEL
LIN {X 0,Y 200.017,Z 523.569,A -85,B 0,C 180,E1 -21503.949,E2 -21503.949} C_VEL
LIN {X 0,Y 200.323,Z 523.53,A -85,B 0,C 180,E1 -21507.989,E2 -21507.989} C_VEL
LIN {X 0,Y 200.472,Z 523.512,A -85,B 0,C 180,E1 -21510,E2 -21510} C_VEL
LIN {X 0,Y 200.019,Z 523.568,A -85,B 0,C 180,E1 -21514.029,E2 -21514.029} C_VEL
LIN {X 0,Y 200.078,Z 523.557,A -85,B 0,C 180,E1 -21518.077,E2 -21518.077} C_VEL
LIN {X 0,Y 199.872,Z 523.586,A -85,B 0,C 180,E1 -21522.179,E2 -21522.179} C_VEL
LIN {X 0,Y 199.798,Z 523.593,A -85,B 0,C 180,E1 -21526.344,E2 -21526.344} C_VEL
LIN {X 0,Y 199.685,Z 523.61,A -85,B 0,C 180,E1 -21530.607,E2 -21530.607} C_VEL
LIN {X 0,Y 199.656,Z 523.613,A -85,B 0,C 180,E1 -21534.987,E2 -21534.987} C_VEL
LIN {X 0,Y 199.612,Z 523.62,A -85,B 0,C 180,E1 -21539.532,E2 -21539.532} C_VEL
LIN {X 0,Y 199.668,Z 523.611,A -85,B 0,C 180,E1 -21542.352,E2 -21542.352} C_VEL
LIN {X 0,Y 199.623,Z 523.617,A -85,B 0,C 180,E1 -21546.763,E2 -21546.763} C_VEL
LIN {X 0,Y 199.6,Z 523.622,A -85,B 0,C 180,E1 -21549.33,E2 -21549.33} C_VEL
LIN {X 0,Y 199.571,Z 523.621,A -85,B 0,C 180,E1 -21552.308,E2 -21552.308} C_VEL
LIN {X 0,Y 199.579,Z 523.625,A -85,B 0,C 180,E1 -21555.227,E2 -21555.227} C_VEL
LIN {X 0,Y 199.58,Z 523.623,A -85,B 0,C 180,E1 -21558.004,E2 -21558.004} C_VEL
LIN {X 0,Y 199.613,Z 523.618,A -85,B 0,C 180,E1 -21560.767,E2 -21560.767} C_VEL
LIN {X 0,Y 199.616,Z 523.619,A -85,B 0,C 180,E1 -21565.713,E2 -21565.713} C_VEL
LIN {X 0,Y 199.703,Z 523.606,A -85,B 0,C 180,E1 -21568.137,E2 -21568.137} C_VEL
LIN {X 0,Y 199.689,Z 523.61,A -85,B 0,C 180,E1 -21572.771,E2 -21572.771} C_VEL
LIN {X 0,Y 199.717,Z 523.605,A -85,B 0,C 180,E1 -21577.226,E2 -21577.226} C_VEL
LIN {X 0,Y 199.798,Z 523.596,A -85,B 0,C 180,E1 -21581.757,E2 -21581.757} C_VEL
LIN {X 0,Y 199.838,Z 523.589,A -85,B 0,C 180,E1 -21585.748,E2 -21585.748} C_VEL
LIN {X 0,Y 200.024,Z 523.567,A -85,B 0,C 180,E1 -21589.881,E2 -21589.881} C_VEL
LIN {X 0,Y 200.014,Z 523.567,A -85,B 0,C 180,E1 -21593.948,E2 -21593.948} C_VEL
LIN {X 0,Y 200.319,Z 523.529,A -85,B 0,C 180,E1 -21597.989,E2 -21597.989} C_VEL
LIN {X 0,Y 200.474,Z 523.511,A -85,B 0,C 180,E1 -21599.999,E2 -21599.999} C_VEL
LIN {X 0,Y 200.008,Z 523.566,A -85,B 0,C 180,E1 -21604.029,E2 -21604.029} C_VEL
LIN {X 0,Y 200.075,Z 523.561,A -85,B 0,C 180,E1 -21608.077,E2 -21608.077} C_VEL
LIN {X 0,Y 199.872,Z 523.584,A -85,B 0,C 180,E1 -21612.179,E2 -21612.179} C_VEL
LIN {X 0,Y 199.79,Z 523.597,A -85,B 0,C 180,E1 -21616.344,E2 -21616.344} C_VEL
LIN {X 0,Y 199.675,Z 523.611,A -85,B 0,C 180,E1 -21620.608,E2 -21620.608} C_VEL
LIN {X 0,Y 199.651,Z 523.616,A -85,B 0,C 180,E1 -21624.987,E2 -21624.987} C_VEL
LIN {X 0,Y 199.609,Z 523.618,A -85,B 0,C 180,E1 -21629.533,E2 -21629.533} C_VEL
LIN {X 0,Y 199.648,Z 523.62,A -85,B 0,C 180,E1 -21632.345,E2 -21632.345} C_VEL
LIN {X 0,Y 199.728,Z 523.665,A -85,B 0,C 180,E1 -21635.165,E2 -21635.165} C_VEL
LIN {X 0,Y 200.834,Z 529.603,A -85,B 0,C 180,E1 -21639.658,E2 -21639.658} C_VEL
LIN {X 0,Y 202.034,Z 535.697,A -85,B 0,C 180,E1 -21644.085,E2 -21644.085} C_VEL
LIN {X 0,Y 203.516,Z 542.873,A -85,B 0,C 180,E1 -21648.995,E2 -21648.995} C_VEL
LIN {X 0,Y 203.809,Z 545.248,A -85,B 0,C 180,E1 -21650.557,E2 -21650.557} C_VEL
LIN {X 0,Y 202.599,Z 550.481,A -85,B 0,C 180,E1 -21653.863,E2 -21653.863} C_VEL
LIN {X 0,Y 200.938,Z 557.694,A -85,B 0,C 180,E1 -21658.356,E2 -21658.356} C_VEL
LIN {X 0,Y 200.573,Z 559.351,A -85,B 0,C 180,E1 -21659.393,E2 -21659.393} C_VEL
LIN {X 0,Y 201.661,Z 574.232,A -85,B 0,C 180,E1 -21660.606,E2 -21660.606} C_VEL
LIN {X 0,Y 202.285,Z 587.095,A -85,B 0,C 180,E1 -21662.029,E2 -21662.029} C_VEL
LIN {X 0,Y 202.654,Z 599.166,A -85,B 0,C 180,E1 -21663.729,E2 -21663.729} C_VEL
LIN {X 0,Y 202.745,Z 610.506,A -85,B 0,C 180,E1 -21665.692,E2 -21665.692} C_VEL
LIN {X 0,Y 202.58,Z 620.699,A -85,B 0,C 180,E1 -21667.835,E2 -21667.835} C_VEL
LIN {X 0,Y 202.204,Z 629.97,A -85,B 0,C 180,E1 -21670.192,E2 -21670.192} C_VEL
LIN {X 0,Y 200.777,Z 638.076,A -85,B 0,C 180,E1 -21672.691,E2 -21672.691} C_VEL
LIN {X 0,Y 199.612,Z 646.045,A -85,B 0,C 180,E1 -21675.732,E2 -21675.732} C_VEL
LIN {X 0,Y 199.082,Z 652.458,A -85,B 0,C 180,E1 -21678.805,E2 -21678.805} C_VEL
LIN {X 0,Y 198.997,Z 655.644,A -85,B 0,C 180,E1 -21680.684,E2 -21680.684} C_VEL
LIN {X 0,Y 198.406,Z 657.905,A -85,B 0,C 180,E1 -21682.249,E2 -21682.249} C_VEL
LIN {X 0,Y 196.977,Z 659.677,A -85,B 0,C 180,E1 -21683.842,E2 -21683.842} C_VEL
LIN {X 0,Y 193.777,Z 662.229,A -85,B 0,C 180,E1 -21687.157,E2 -21687.157} C_VEL
LIN {X 0,Y 193.08,Z 663.258,A -85,B 0,C 180,E1 -21688.893,E2 -21688.893} C_VEL
LIN {X 0,Y 193.12,Z 663.558,A -85,B 0,C 180,E1 -21689.475,E2 -21689.475} C_VEL
LIN {X 0,Y 193.238,Z 663.876,A -85,B 0,C 180,E1 -21690,E2 -21690} C_VEL
LIN {X 0,Y 192.633,Z 664.479,A -85,B 0,C 180,E1 -21692.091,E2 -21692.091} C_VEL
LIN {X 0,Y 191.721,Z 664.474,A -85,B 0,C 180,E1 -21696.314,E2 -21696.314} C_VEL
LIN {X 0,Y 191.303,Z 662.895,A -85,B 0,C 180,E1 -21700.585,E2 -21700.585} C_VEL
LIN {X 0,Y 192.068,Z 659.794,A -85,B 0,C 180,E1 -21704.841,E2 -21704.841} C_VEL
LIN {X 0,Y 193.992,Z 655.218,A -85,B 0,C 180,E1 -21709.03,E2 -21709.03} C_VEL
LIN {X 0,Y 196.388,Z 650.688,A -85,B 0,C 180,E1 -21712.071,E2 -21712.071} C_VEL
LIN {X 0,Y 200.037,Z 644.115,A -85,B 0,C 180,E1 -21715.492,E2 -21715.492} C_VEL
LIN {X 0,Y 203.247,Z 637.256,A -85,B 0,C 180,E1 -21718.389,E2 -21718.389} C_VEL
LIN {X 0,Y 207.04,Z 628.276,A -85,B 0,C 180,E1 -21721.474,E2 -21721.474} C_VEL
LIN {X 0,Y 210.104,Z 619.415,A -85,B 0,C 180,E1 -21724.076,E2 -21724.076} C_VEL
LIN {X 0,Y 212.836,Z 608.202,A -85,B 0,C 180,E1 -21727.065,E2 -21727.065} C_VEL
LIN {X 0,Y 214.459,Z 597.591,A -85,B 0,C 180,E1 -21729.716,E2 -21729.716} C_VEL
LIN {X 0,Y 215.304,Z 586.457,A -85,B 0,C 180,E1 -21732.452,E2 -21732.452} C_VEL
LIN {X 0,Y 215.333,Z 577.052,A -85,B 0,C 180,E1 -21734.885,E2 -21734.885} C_VEL
LIN {X 0,Y 214.33,Z 572.641,A -85,B 0,C 180,E1 -21736.481,E2 -21736.481} C_VEL
LIN {X 0,Y 212.179,Z 565.587,A -85,B 0,C 180,E1 -21739.626,E2 -21739.626} C_VEL
LIN {X 0,Y 209.602,Z 557.334,A -85,B 0,C 180,E1 -21744.328,E2 -21744.328} C_VEL
LIN {X 0,Y 207.602,Z 552.299,A -85,B 0,C 180,E1 -21749.483,E2 -21749.483} C_VEL
LIN {X 0,Y 207.349,Z 549.475,A -85,B 0,C 180,E1 -21753.856,E2 -21753.856} C_VEL
LIN {X 0,Y 208.4,Z 548.061,A -85,B 0,C 180,E1 -21758.226,E2 -21758.226} C_VEL
LIN {X 0,Y 211.495,Z 549.927,A -85,B 0,C 180,E1 -21764.584,E2 -21764.584} C_VEL
LIN {X 0,Y 213.461,Z 552.641,A -85,B 0,C 180,E1 -21767.654,E2 -21767.654} C_VEL
LIN {X 0,Y 215.707,Z 558.342,A -85,B 0,C 180,E1 -21771.57,E2 -21771.57} C_VEL
LIN {X 0,Y 217.908,Z 564.428,A -85,B 0,C 180,E1 -21775.2,E2 -21775.2} C_VEL
LIN {X 0,Y 219.048,Z 570.505,A -85,B 0,C 180,E1 -21778.162,E2 -21778.162} C_VEL
LIN {X 0,Y 219.789,Z 577.323,A -85,B 0,C 180,E1 -21781.375,E2 -21781.375} C_VEL
LIN {X 0,Y 219.754,Z 581.229,A -85,B 0,C 180,E1 -21783.131,E2 -21783.131} C_VEL
LIN {X 0,Y 219.497,Z 582.595,A -85,B 0,C 180,E1 -21783.672,E2 -21783.672} C_VEL
LIN {X 0,Y 215.351,Z 590.033,A -85,B 0,C 180,E1 -21786.089,E2 -21786.089} C_VEL
LIN {X 0,Y 210.742,Z 597.284,A -85,B 0,C 180,E1 -21789.115,E2 -21789.115} C_VEL
LIN {X 0,Y 207.275,Z 602.084,A -85,B 0,C 180,E1 -21791.739,E2 -21791.739} C_VEL
LIN {X 0,Y 203.662,Z 606.455,A -85,B 0,C 180,E1 -21794.931,E2 -21794.931} C_VEL
LIN {X 0,Y 200.23,Z 609.799,A -85,B 0,C 180,E1 -21798.612,E2 -21798.612} C_VEL
LIN {X 0,Y 197.535,Z 611.709,A -85,B 0,C 180,E1 -21802.324,E2 -21802.324} C_VEL
LIN {X 0,Y 195.531,Z 612.278,A -85,B 0,C 180,E1 -21806.027,E2 -21806.027} C_VEL
LIN {X 0,Y 194.145,Z 611.582,A -85,B 0,C 180,E1 -21809.68,E2 -21809.68} C_VEL
LIN {X 0,Y 193.395,Z 609.715,A -85,B 0,C 180,E1 -21813.297,E2 -21813.297} C_VEL
LIN {X 0,Y 193.156,Z 606.753,A -85,B 0,C 180,E1 -21816.824,E2 -21816.824} C_VEL
LIN {X 0,Y 193.391,Z 602.702,A -85,B 0,C 180,E1 -21820.256,E2 -21820.256} C_VEL
LIN {X 0,Y 194.117,Z 597.5,A -85,B 0,C 180,E1 -21823.605,E2 -21823.605} C_VEL
LIN {X 0,Y 195.231,Z 591.09,A -85,B 0,C 180,E1 -21826.845,E2 -21826.845} C_VEL
LIN {X 0,Y 196.694,Z 582.767,A -85,B 0,C 180,E1 -21830.189,E2 -21830.189} C_VEL
LIN {X 0,Y 198.341,Z 574.205,A -85,B 0,C 180,E1 -21832.959,E2 -21832.959} C_VEL
LIN {X 0,Y 200.187,Z 564.382,A -85,B 0,C 180,E1 -21835.529,E2 -21835.529} C_VEL
LIN {X 0,Y 201.534,Z 556.281,A -85,B 0,C 180,E1 -21837.302,E2 -21837.302} C_VEL
LIN {X 0,Y 199.924,Z 548.641,A -85,B 0,C 180,E1 -21838.988,E2 -21838.988} C_VEL
LIN {X 0,Y 196.732,Z 537.38,A -85,B 0,C 180,E1 -21841.226,E2 -21841.226} C_VEL
LIN {X 0,Y 192.949,Z 525.839,A -85,B 0,C 180,E1 -21843.208,E2 -21843.208} C_VEL
LIN {X 0,Y 192.635,Z 524.493,A -85,B 0,C 180,E1 -21843.453,E2 -21843.453} C_VEL
LIN {X 0,Y 192.689,Z 524.482,A -85,B 0,C 180,E1 -21846.346,E2 -21846.346} C_VEL
LIN {X 0,Y 192.734,Z 524.48,A -85,B 0,C 180,E1 -21851.459,E2 -21851.459} C_VEL
LIN {X 0,Y 192.756,Z 524.477,A -85,B 0,C 180,E1 -21855.213,E2 -21855.213} C_VEL
LIN {X 0,Y 192.949,Z 524.452,A -85,B 0,C 180,E1 -21859.567,E2 -21859.567} C_VEL
LIN {X 0,Y 192.98,Z 524.447,A -85,B 0,C 180,E1 -21863.727,E2 -21863.727} C_VEL
LIN {X 0,Y 193.264,Z 524.409,A -85,B 0,C 180,E1 -21867.916,E2 -21867.916} C_VEL
LIN {X 0,Y 193.437,Z 524.388,A -85,B 0,C 180,E1 -21870,E2 -21870} C_VEL
LIN {X 0,Y 192.965,Z 524.447,A -85,B 0,C 180,E1 -21874.177,E2 -21874.177} C_VEL
LIN {X 0,Y 193.029,Z 524.435,A -85,B 0,C 180,E1 -21878.374,E2 -21878.374} C_VEL
LIN {X 0,Y 192.799,Z 524.468,A -85,B 0,C 180,E1 -21882.633,E2 -21882.633} C_VEL
LIN {X 0,Y 192.755,Z 524.472,A -85,B 0,C 180,E1 -21886.959,E2 -21886.959} C_VEL
LIN {X 0,Y 192.618,Z 524.492,A -85,B 0,C 180,E1 -21891.399,E2 -21891.399} C_VEL
LIN {X 0,Y 192.644,Z 524.485,A -85,B 0,C 180,E1 -21894.208,E2 -21894.208} C_VEL
LIN {X 0,Y 192.606,Z 524.492,A -85,B 0,C 180,E1 -21898.866,E2 -21898.866} C_VEL
LIN {X 0,Y 192.597,Z 524.492,A -85,B 0,C 180,E1 -21903.186,E2 -21903.186} C_VEL
LIN {X 0,Y 192.547,Z 524.499,A -85,B 0,C 180,E1 -21908.353,E2 -21908.353} C_VEL
LIN {X 0,Y 192.489,Z 524.505,A -85,B 0,C 180,E1 -21913.094,E2 -21913.094} C_VEL
LIN {X 0,Y 192.492,Z 524.508,A -85,B 0,C 180,E1 -21916.904,E2 -21916.904} C_VEL
LIN {X 0,Y 192.553,Z 524.495,A -85,B 0,C 180,E1 -21921.648,E2 -21921.648} C_VEL
LIN {X 0,Y 192.601,Z 524.494,A -85,B 0,C 180,E1 -21926.814,E2 -21926.814} C_VEL
LIN {X 0,Y 192.667,Z 524.483,A -85,B 0,C 180,E1 -21931.691,E2 -21931.691} C_VEL
LIN {X 0,Y 192.687,Z 524.481,A -85,B 0,C 180,E1 -21936.345,E2 -21936.345} C_VEL
LIN {X 0,Y 192.734,Z 524.476,A -85,B 0,C 180,E1 -21941.457,E2 -21941.457} C_VEL
LIN {X 0,Y 192.766,Z 524.471,A -85,B 0,C 180,E1 -21945.213,E2 -21945.213} C_VEL
LIN {X 0,Y 192.947,Z 524.449,A -85,B 0,C 180,E1 -21949.566,E2 -21949.566} C_VEL
LIN {X 0,Y 192.977,Z 524.444,A -85,B 0,C 180,E1 -21953.727,E2 -21953.727} C_VEL
LIN {X 0,Y 193.26,Z 524.409,A -85,B 0,C 180,E1 -21957.915,E2 -21957.915} C_VEL
LIN {X 0,Y 193.438,Z 524.388,A -85,B 0,C 180,E1 -21959.999,E2 -21959.999} C_VEL
LIN {X 0,Y 192.954,Z 524.445,A -85,B 0,C 180,E1 -21964.177,E2 -21964.177} C_VEL
LIN {X 0,Y 193.026,Z 524.44,A -85,B 0,C 180,E1 -21968.374,E2 -21968.374} C_VEL
LIN {X 0,Y 192.798,Z 524.466,A -85,B 0,C 180,E1 -21972.633,E2 -21972.633} C_VEL
LIN {X 0,Y 192.748,Z 524.477,A -85,B 0,C 180,E1 -21976.959,E2 -21976.959} C_VEL
LIN {X 0,Y 192.609,Z 524.488,A -85,B 0,C 180,E1 -21981.4,E2 -21981.4} C_VEL
LIN {X 0,Y 192.64,Z 524.487,A -85,B 0,C 180,E1 -21984.208,E2 -21984.208} C_VEL
LIN {X 0,Y 192.602,Z 524.492,A -85,B 0,C 180,E1 -21988.866,E2 -21988.866} C_VEL
LIN {X 0,Y 192.651,Z 524.531,A -85,B 0,C 180,E1 -21994.75,E2 -21994.75} C_VEL
LIN {X 0,Y 193.751,Z 530.318,A -85,B 0,C 180,E1 -21999.311,E2 -21999.311} C_VEL
LIN {X 0,Y 194.958,Z 536.392,A -85,B 0,C 180,E1 -22003.865,E2 -22003.865} C_VEL
LIN {X 0,Y 196.378,Z 543.26,A -85,B 0,C 180,E1 -22008.724,E2 -22008.724} C_VEL
LIN {X 0,Y 196.566,Z 546.768,A -85,B 0,C 180,E1 -22011.106,E2 -22011.106} C_VEL
LIN {X 0,Y 194.612,Z 554.504,A -85,B 0,C 180,E1 -22016.16,E2 -22016.16} C_VEL
LIN {X 0,Y 193.713,Z 558.316,A -85,B 0,C 180,E1 -22018.641,E2 -22018.641} C_VEL
LIN {X 0,Y 194.766,Z 573.971,A -85,B 0,C 180,E1 -22019.999,E2 -22019.999} C_VEL
LIN {X 0,Y 195.37,Z 587.687,A -85,B 0,C 180,E1 -22021.621,E2 -22021.621} C_VEL
LIN {X 0,Y 195.665,Z 598.632,A -85,B 0,C 180,E1 -22023.252,E2 -22023.252} C_VEL
LIN {X 0,Y 195.69,Z 610.063,A -85,B 0,C 180,E1 -22025.323,E2 -22025.323} C_VEL
LIN {X 0,Y 195.521,Z 620.133,A -85,B 0,C 180,E1 -22027.548,E2 -22027.548} C_VEL
LIN {X 0,Y 195.265,Z 627.835,A -85,B 0,C 180,E1 -22029.555,E2 -22029.555} C_VEL
LIN {X 0,Y 194.018,Z 635.931,A -85,B 0,C 180,E1 -22032.068,E2 -22032.068} C_VEL
LIN {X 0,Y 192.628,Z 644.05,A -85,B 0,C 180,E1 -22035.203,E2 -22035.203} C_VEL
LIN {X 0,Y 192.078,Z 650.649,A -85,B 0,C 180,E1 -22038.391,E2 -22038.391} C_VEL
LIN {X 0,Y 192.002,Z 655.855,A -85,B 0,C 180,E1 -22041.581,E2 -22041.581} C_VEL
LIN {X 0,Y 192.418,Z 659.835,A -85,B 0,C 180,E1 -22044.761,E2 -22044.761} C_VEL
LIN {X 0,Y 192.864,Z 662.613,A -85,B 0,C 180,E1 -22047.912,E2 -22047.912} C_VEL
LIN {X 0,Y 193.12,Z 663.558,A -85,B 0,C 180,E1 -22049.475,E2 -22049.475} C_VEL
LIN {X 0,Y 192.908,Z 664.094,A -85,B 0,C 180,E1 -22050.618,E2 -22050.618} C_VEL
LIN {X 0,Y 192.003,Z 664.36,A -85,B 0,C 180,E1 -22051.748,E2 -22051.748} C_VEL
LIN {X 0,Y 189.062,Z 664.273,A -85,B 0,C 180,E1 -22053.968,E2 -22053.968} C_VEL
LIN {X 0,Y 185.9,Z 663.645,A -85,B 0,C 180,E1 -22056.269,E2 -22056.269} C_VEL
LIN {X 0,Y 184.459,Z 663.05,A -85,B 0,C 180,E1 -22058.088,E2 -22058.088} C_VEL
LIN {X 0,Y 184.309,Z 662.844,A -85,B 0,C 180,E1 -22058.714,E2 -22058.714} C_VEL
LIN {X 0,Y 184.556,Z 660.677,A -85,B 0,C 180,E1 -22063.208,E2 -22063.208} C_VEL
LIN {X 0,Y 186.038,Z 657.013,A -85,B 0,C 180,E1 -22067.591,E2 -22067.591} C_VEL
LIN {X 0,Y 187.958,Z 653.262,A -85,B 0,C 180,E1 -22070.808,E2 -22070.808} C_VEL
LIN {X 0,Y 191.856,Z 646.828,A -85,B 0,C 180,E1 -22074.915,E2 -22074.915} C_VEL
LIN {X 0,Y 195.303,Z 640.767,A -85,B 0,C 180,E1 -22077.892,E2 -22077.892} C_VEL
LIN {X 0,Y 199.394,Z 632.189,A -85,B 0,C 180,E1 -22081.325,E2 -22081.325} C_VEL
LIN {X 0,Y 203.138,Z 623.421,A -85,B 0,C 180,E1 -22084.209,E2 -22084.209} C_VEL
LIN {X 0,Y 206.26,Z 613.16,A -85,B 0,C 180,E1 -22087.215,E2 -22087.215} C_VEL
LIN {X 0,Y 208.474,Z 603.527,A -85,B 0,C 180,E1 -22089.831,E2 -22089.831} C_VEL
LIN {X 0,Y 210.142,Z 591.619,A -85,B 0,C 180,E1 -22092.98,E2 -22092.98} C_VEL
LIN {X 0,Y 210.768,Z 582.147,A -85,B 0,C 180,E1 -22095.554,E2 -22095.554} C_VEL
LIN {X 0,Y 210.363,Z 578.753,A -85,B 0,C 180,E1 -22096.775,E2 -22096.775} C_VEL
LIN {X 0,Y 208.54,Z 571.299,A -85,B 0,C 180,E1 -22100.185,E2 -22100.185} C_VEL
LIN {X 0,Y 206.527,Z 563.582,A -85,B 0,C 180,E1 -22104.757,E2 -22104.757} C_VEL
LIN {X 0,Y 205.011,Z 559.407,A -85,B 0,C 180,E1 -22109.055,E2 -22109.055} C_VEL
LIN {X 0,Y 204.688,Z 556.483,A -85,B 0,C 180,E1 -22113.217,E2 -22113.217} C_VEL
LIN {X 0,Y 205.525,Z 554.744,A -85,B 0,C 180,E1 -22117.905,E2 -22117.905} C_VEL
LIN {X 0,Y 206.202,Z 554.96,A -85,B 0,C 180,E1 -22120.073,E2 -22120.073} C_VEL
LIN {X 0,Y 208.245,Z 556.262,A -85,B 0,C 180,E1 -22124.337,E2 -22124.337} C_VEL
LIN {X 0,Y 209.889,Z 558.808,A -85,B 0,C 180,E1 -22127.441,E2 -22127.441} C_VEL
LIN {X 0,Y 211.636,Z 564.24,A -85,B 0,C 180,E1 -22131.406,E2 -22131.406} C_VEL
LIN {X 0,Y 213.352,Z 570.399,A -85,B 0,C 180,E1 -22135.277,E2 -22135.277} C_VEL
LIN {X 0,Y 214.108,Z 577.685,A -85,B 0,C 180,E1 -22139.06,E2 -22139.06} C_VEL
LIN {X 0,Y 214.09,Z 583.281,A -85,B 0,C 180,E1 -22141.882,E2 -22141.882} C_VEL
LIN {X 0,Y 213.635,Z 585.431,A -85,B 0,C 180,E1 -22142.829,E2 -22142.829} C_VEL
LIN {X 0,Y 208.462,Z 593.911,A -85,B 0,C 180,E1 -22145.805,E2 -22145.805} C_VEL
LIN {X 0,Y 203.703,Z 600.537,A -85,B 0,C 180,E1 -22148.932,E2 -22148.932} C_VEL
LIN {X 0,Y 199.451,Z 605.681,A -85,B 0,C 180,E1 -22152.206,E2 -22152.206} C_VEL
LIN {X 0,Y 196.424,Z 608.827,A -85,B 0,C 180,E1 -22154.97,E2 -22154.97} C_VEL
LIN {X 0,Y 192.984,Z 611.719,A -85,B 0,C 180,E1 -22158.761,E2 -22158.761} C_VEL
LIN {X 0,Y 190.289,Z 613.152,A -85,B 0,C 180,E1 -22162.58,E2 -22162.58} C_VEL
LIN {X 0,Y 188.217,Z 613.293,A -85,B 0,C 180,E1 -22166.621,E2 -22166.621} C_VEL
LIN {X 0,Y 186.956,Z 612.285,A -85,B 0,C 180,E1 -22170.161,E2 -22170.161} C_VEL
LIN {X 0,Y 186.228,Z 609.616,A -85,B 0,C 180,E1 -22174.478,E2 -22174.478} C_VEL
LIN {X 0,Y 186.18,Z 605.57,A -85,B 0,C 180,E1 -22178.619,E2 -22178.619} C_VEL
LIN {X 0,Y 186.791,Z 600.055,A -85,B 0,C 180,E1 -22182.63,E2 -22182.63} C_VEL
LIN {X 0,Y 187.777,Z 594.001,A -85,B 0,C 180,E1 -22186.004,E2 -22186.004} C_VEL
LIN {X 0,Y 189.284,Z 585.942,A -85,B 0,C 180,E1 -22189.567,E2 -22189.567} C_VEL
LIN {X 0,Y 191.016,Z 576.922,A -85,B 0,C 180,E1 -22192.716,E2 -22192.716} C_VEL
LIN {X 0,Y 193.004,Z 566.711,A -85,B 0,C 180,E1 -22195.586,E2 -22195.586} C_VEL
LIN {X 0,Y 194.605,Z 556.955,A -85,B 0,C 180,E1 -22197.812,E2 -22197.812} C_VEL
LIN {X 0,Y 192.456,Z 548.063,A -85,B 0,C 180,E1 -22199.86,E2 -22199.86} C_VEL
LIN {X 0,Y 189.393,Z 537.169,A -85,B 0,C 180,E1 -22202.063,E2 -22202.063} C_VEL
LIN {X 0,Y 185.553,Z 525.373,A -85,B 0,C 180,E1 -22204.179,E2 -22204.179} C_VEL
LIN {X 0,Y 185.579,Z 525.369,A -85,B 0,C 180,E1 -22207.746,E2 -22207.746} C_VEL
LIN {X 0,Y 185.688,Z 525.355,A -85,B 0,C 180,E1 -22212.375,E2 -22212.375} C_VEL
LIN {X 0,Y 185.727,Z 525.351,A -85,B 0,C 180,E1 -22216.877,E2 -22216.877} C_VEL
LIN {X 0,Y 185.981,Z 525.32,A -85,B 0,C 180,E1 -22221.306,E2 -22221.306} C_VEL
LIN {X 0,Y 186.208,Z 525.289,A -85,B 0,C 180,E1 -22227.837,E2 -22227.837} C_VEL
LIN {X 0,Y 186.402,Z 525.265,A -85,B 0,C 180,E1 -22230,E2 -22230} C_VEL
LIN {X 0,Y 185.912,Z 525.326,A -85,B 0,C 180,E1 -22234.336,E2 -22234.336} C_VEL
LIN {X 0,Y 185.978,Z 525.314,A -85,B 0,C 180,E1 -22238.694,E2 -22238.694} C_VEL
LIN {X 0,Y 185.726,Z 525.351,A -85,B 0,C 180,E1 -22243.123,E2 -22243.123} C_VEL
LIN {X 0,Y 185.69,Z 525.351,A -85,B 0,C 180,E1 -22247.625,E2 -22247.625} C_VEL
LIN {X 0,Y 185.579,Z 525.367,A -85,B 0,C 180,E1 -22252.253,E2 -22252.253} C_VEL
LIN {X 0,Y 185.513,Z 525.373,A -85,B 0,C 180,E1 -22257.04,E2 -22257.04} C_VEL
LIN {X 0,Y 185.547,Z 525.373,A -85,B 0,C 180,E1 -22259.499,E2 -22259.499} C_VEL
LIN {X 0,Y 185.5,Z 525.373,A -85,B 0,C 180,E1 -22264.632,E2 -22264.632} C_VEL
LIN {X 0,Y 185.504,Z 525.379,A -85,B 0,C 180,E1 -22267.313,E2 -22267.313} C_VEL
LIN {X 0,Y 185.466,Z 525.382,A -85,B 0,C 180,E1 -22270.722,E2 -22270.722} C_VEL
LIN {X 0,Y 185.461,Z 525.381,A -85,B 0,C 180,E1 -22276.055,E2 -22276.055} C_VEL
LIN {X 0,Y 185.47,Z 525.378,A -85,B 0,C 180,E1 -22279.895,E2 -22279.895} C_VEL
LIN {X 0,Y 185.508,Z 525.373,A -85,B 0,C 180,E1 -22282.711,E2 -22282.711} C_VEL
LIN {X 0,Y 185.549,Z 525.369,A -85,B 0,C 180,E1 -22287.975,E2 -22287.975} C_VEL
LIN {X 0,Y 185.584,Z 525.362,A -85,B 0,C 180,E1 -22290.575,E2 -22290.575} C_VEL
LIN {X 0,Y 185.582,Z 525.367,A -85,B 0,C 180,E1 -22295.381,E2 -22295.381} C_VEL
LIN {X 0,Y 185.676,Z 525.357,A -85,B 0,C 180,E1 -22301.133,E2 -22301.133} C_VEL
LIN {X 0,Y 185.697,Z 525.353,A -85,B 0,C 180,E1 -22304.637,E2 -22304.637} C_VEL
LIN {X 0,Y 185.889,Z 525.329,A -85,B 0,C 180,E1 -22309.418,E2 -22309.418} C_VEL
LIN {X 0,Y 185.94,Z 525.321,A -85,B 0,C 180,E1 -22313.489,E2 -22313.489} C_VEL
LIN {X 0,Y 186.204,Z 525.288,A -85,B 0,C 180,E1 -22317.836,E2 -22317.836} C_VEL
LIN {X 0,Y 186.402,Z 525.264,A -85,B 0,C 180,E1 -22319.999,E2 -22319.999} C_VEL
LIN {X 0,Y 185.901,Z 525.323,A -85,B 0,C 180,E1 -22324.336,E2 -22324.336} C_VEL
LIN {X 0,Y 185.975,Z 525.32,A -85,B 0,C 180,E1 -22328.694,E2 -22328.694} C_VEL
LIN {X 0,Y 185.724,Z 525.347,A -85,B 0,C 180,E1 -22333.123,E2 -22333.123} C_VEL
LIN {X 0,Y 185.685,Z 525.354,A -85,B 0,C 180,E1 -22337.625,E2 -22337.625} C_VEL
LIN {X 0,Y 185.572,Z 525.364,A -85,B 0,C 180,E1 -22342.254,E2 -22342.254} C_VEL
LIN {X 0,Y 185.577,Z 525.368,A -85,B 0,C 180,E1 -22344.646,E2 -22344.646} C_VEL
LIN {X 0,Y 185.544,Z 525.37,A -85,B 0,C 180,E1 -22349.499,E2 -22349.499} C_VEL
LIN {X 0,Y 185.599,Z 525.534,A -85,B 0,C 180,E1 -22354.454,E2 -22354.454} C_VEL
LIN {X 0,Y 186.579,Z 530.542,A -85,B 0,C 180,E1 -22358.56,E2 -22358.56} C_VEL
LIN {X 0,Y 187.844,Z 537.04,A -85,B 0,C 180,E1 -22363.606,E2 -22363.606} C_VEL
LIN {X 0,Y 189.315,Z 544.007,A -85,B 0,C 180,E1 -22368.755,E2 -22368.755} C_VEL
LIN {X 0,Y 189.396,Z 547.472,A -85,B 0,C 180,E1 -22371.192,E2 -22371.192} C_VEL
LIN {X 0,Y 187.61,Z 554.315,A -85,B 0,C 180,E1 -22375.812,E2 -22375.812} C_VEL
LIN {X 0,Y 186.836,Z 557.406,A -85,B 0,C 180,E1 -22377.905,E2 -22377.905} C_VEL
LIN {X 0,Y 187.845,Z 572.391,A -85,B 0,C 180,E1 -22379.231,E2 -22379.231} C_VEL
LIN {X 0,Y 188.384,Z 585.458,A -85,B 0,C 180,E1 -22380.795,E2 -22380.795} C_VEL
LIN {X 0,Y 188.664,Z 598.767,A -85,B 0,C 180,E1 -22382.851,E2 -22382.851} C_VEL
LIN {X 0,Y 188.665,Z 609.6,A -85,B 0,C 180,E1 -22384.93,E2 -22384.93} C_VEL
LIN {X 0,Y 188.486,Z 619.574,A -85,B 0,C 180,E1 -22387.242,E2 -22387.242} C_VEL
LIN {X 0,Y 188.044,Z 629.23,A -85,B 0,C 180,E1 -22389.943,E2 -22389.943} C_VEL
LIN {X 0,Y 186.412,Z 638.132,A -85,B 0,C 180,E1 -22393.011,E2 -22393.011} C_VEL
LIN {X 0,Y 185.42,Z 645.665,A -85,B 0,C 180,E1 -22396.297,E2 -22396.297} C_VEL
LIN {X 0,Y 184.981,Z 652.581,A -85,B 0,C 180,E1 -22400.157,E2 -22400.157} C_VEL
LIN {X 0,Y 185.162,Z 657.096,A -85,B 0,C 180,E1 -22403.462,E2 -22403.462} C_VEL
LIN {X 0,Y 185.491,Z 659.417,A -85,B 0,C 180,E1 -22405.654,E2 -22405.654} C_VEL
LIN {X 0,Y 185.832,Z 661.223,A -85,B 0,C 180,E1 -22407.833,E2 -22407.833} C_VEL
LIN {X 0,Y 186.248,Z 662.572,A -85,B 0,C 180,E1 -22410,E2 -22410} C_VEL
LIN {X 0,Y 185.596,Z 663.257,A -85,B 0,C 180,E1 -22412.17,E2 -22412.17} C_VEL
LIN {X 0,Y 184.653,Z 663.367,A -85,B 0,C 180,E1 -22416.557,E2 -22416.557} C_VEL
LIN {X 0,Y 184.309,Z 662.844,A -85,B 0,C 180,E1 -22418.714,E2 -22418.714} C_VEL
LIN {X 0,Y 183.599,Z 662.133,A -85,B 0,C 180,E1 -22420.528,E2 -22420.528} C_VEL
LIN {X 0,Y 181.051,Z 660.383,A -85,B 0,C 180,E1 -22423.493,E2 -22423.493} C_VEL
LIN {X 0,Y 179.054,Z 658.006,A -85,B 0,C 180,E1 -22426.492,E2 -22426.492} C_VEL
LIN {X 0,Y 179.217,Z 656.315,A -85,B 0,C 180,E1 -22428.301,E2 -22428.301} C_VEL
LIN {X 0,Y 181.079,Z 653.075,A -85,B 0,C 180,E1 -22431.333,E2 -22431.333} C_VEL
LIN {X 0,Y 184.293,Z 648.257,A -85,B 0,C 180,E1 -22434.802,E2 -22434.802} C_VEL
LIN {X 0,Y 188.423,Z 641.752,A -85,B 0,C 180,E1 -22438.396,E2 -22438.396} C_VEL
LIN {X 0,Y 192.665,Z 633.738,A -85,B 0,C 180,E1 -22441.934,E2 -22441.934} C_VEL
LIN {X 0,Y 196.628,Z 625.501,A -85,B 0,C 180,E1 -22444.882,E2 -22444.882} C_VEL
LIN {X 0,Y 200.106,Z 615.99,A -85,B 0,C 180,E1 -22447.925,E2 -22447.925} C_VEL
LIN {X 0,Y 202.735,Z 606.684,A -85,B 0,C 180,E1 -22450.636,E2 -22450.636} C_VEL
LIN {X 0,Y 205.003,Z 595.059,A -85,B 0,C 180,E1 -22453.951,E2 -22453.951} C_VEL
LIN {X 0,Y 206.063,Z 586.404,A -85,B 0,C 180,E1 -22456.451,E2 -22456.451} C_VEL
LIN {X 0,Y 205.944,Z 583.892,A -85,B 0,C 180,E1 -22457.393,E2 -22457.393} C_VEL
LIN {X 0,Y 204.819,Z 577.82,A -85,B 0,C 180,E1 -22460.254,E2 -22460.254} C_VEL
LIN {X 0,Y 203.159,Z 570.062,A -85,B 0,C 180,E1 -22464.975,E2 -22464.975} C_VEL
LIN {X 0,Y 202.339,Z 567.443,A -85,B 0,C 180,E1 -22467.37,E2 -22467.37} C_VEL
LIN {X 0,Y 201.691,Z 564.557,A -85,B 0,C 180,E1 -22470.802,E2 -22470.802} C_VEL
LIN {X 0,Y 201.795,Z 562.23,A -85,B 0,C 180,E1 -22474.894,E2 -22474.894} C_VEL
LIN {X 0,Y 202.376,Z 561.312,A -85,B 0,C 180,E1 -22477.543,E2 -22477.543} C_VEL
LIN {X 0,Y 202.99,Z 561.29,A -85,B 0,C 180,E1 -22479.744,E2 -22479.744} C_VEL
LIN {X 0,Y 204.72,Z 562.423,A -85,B 0,C 180,E1 -22484.06,E2 -22484.06} C_VEL
LIN {X 0,Y 205.646,Z 563.788,A -85,B 0,C 180,E1 -22486.16,E2 -22486.16} C_VEL
LIN {X 0,Y 206.349,Z 566.005,A -85,B 0,C 180,E1 -22488.209,E2 -22488.209} C_VEL
LIN {X 0,Y 207.579,Z 571.351,A -85,B 0,C 180,E1 -22492.217,E2 -22492.217} C_VEL
LIN {X 0,Y 208.479,Z 575.808,A -85,B 0,C 180,E1 -22495.166,E2 -22495.166} C_VEL
LIN {X 0,Y 208.643,Z 582.704,A -85,B 0,C 180,E1 -22499.035,E2 -22499.035} C_VEL
LIN {X 0,Y 208.308,Z 587.141,A -85,B 0,C 180,E1 -22501.45,E2 -22501.45} C_VEL
LIN {X 0,Y 207.856,Z 588.314,A -85,B 0,C 180,E1 -22501.938,E2 -22501.938} C_VEL
LIN {X 0,Y 202.395,Z 596.378,A -85,B 0,C 180,E1 -22504.981,E2 -22504.981} C_VEL
LIN {X 0,Y 197.433,Z 602.772,A -85,B 0,C 180,E1 -22508.187,E2 -22508.187} C_VEL
LIN {X 0,Y 193.429,Z 607.173,A -85,B 0,C 180,E1 -22511.18,E2 -22511.18} C_VEL
LIN {X 0,Y 189.121,Z 611.108,A -85,B 0,C 180,E1 -22515.078,E2 -22515.078} C_VEL
LIN {X 0,Y 185.731,Z 613.476,A -85,B 0,C 180,E1 -22518.914,E2 -22518.914} C_VEL
LIN {X 0,Y 183.049,Z 614.508,A -85,B 0,C 180,E1 -22522.859,E2 -22522.859} C_VEL
LIN {X 0,Y 181.064,Z 614.269,A -85,B 0,C 180,E1 -22526.779,E2 -22526.779} C_VEL
LIN {X 0,Y 179.771,Z 612.861,A -85,B 0,C 180,E1 -22530.674,E2 -22530.674} C_VEL
LIN {X 0,Y 179.179,Z 610.302,A -85,B 0,C 180,E1 -22534.543,E2 -22534.543} C_VEL
LIN {X 0,Y 179.125,Z 606.003,A -85,B 0,C 180,E1 -22538.886,E2 -22538.886} C_VEL
LIN {X 0,Y 179.837,Z 600.056,A -85,B 0,C 180,E1 -22543.171,E2 -22543.171} C_VEL
LIN {X 0,Y 180.997,Z 593.219,A -85,B 0,C 180,E1 -22546.94,E2 -22546.94} C_VEL
LIN {X 0,Y 182.51,Z 585.334,A -85,B 0,C 180,E1 -22550.369,E2 -22550.369} C_VEL
LIN {X 0,Y 184.413,Z 576.036,A -85,B 0,C 180,E1 -22553.619,E2 -22553.619} C_VEL
LIN {X 0,Y 186.471,Z 565.499,A -85,B 0,C 180,E1 -22556.534,E2 -22556.534} C_VEL
LIN {X 0,Y 187.613,Z 559.003,A -85,B 0,C 180,E1 -22558.053,E2 -22558.053} C_VEL
LIN {X 0,Y 187.12,Z 555.466,A -85,B 0,C 180,E1 -22558.906,E2 -22558.906} C_VEL
LIN {X 0,Y 184.258,Z 544.621,A -85,B 0,C 180,E1 -22561.4,E2 -22561.4} C_VEL
LIN {X 0,Y 181.079,Z 534.109,A -85,B 0,C 180,E1 -22563.491,E2 -22563.491} C_VEL
LIN {X 0,Y 178.522,Z 526.25,A -85,B 0,C 180,E1 -22564.887,E2 -22564.887} C_VEL
LIN {X 0,Y 178.624,Z 526.235,A -85,B 0,C 180,E1 -22570.787,E2 -22570.787} C_VEL
LIN {X 0,Y 178.655,Z 526.231,A -85,B 0,C 180,E1 -22576.347,E2 -22576.347} C_VEL
LIN {X 0,Y 178.91,Z 526.2,A -85,B 0,C 180,E1 -22580.959,E2 -22580.959} C_VEL
LIN {X 0,Y 179.153,Z 526.168,A -85,B 0,C 180,E1 -22587.751,E2 -22587.751} C_VEL
LIN {X 0,Y 179.366,Z 526.141,A -85,B 0,C 180,E1 -22590,E2 -22590} C_VEL
LIN {X 0,Y 178.859,Z 526.204,A -85,B 0,C 180,E1 -22594.507,E2 -22594.507} C_VEL
LIN {X 0,Y 178.909,Z 526.195,A -85,B 0,C 180,E1 -22599.04,E2 -22599.04} C_VEL
LIN {X 0,Y 178.655,Z 526.23,A -85,B 0,C 180,E1 -22603.652,E2 -22603.652} C_VEL
LIN {X 0,Y 178.624,Z 526.233,A -85,B 0,C 180,E1 -22609.213,E2 -22609.213} C_VEL
LIN {X 0,Y 178.518,Z 526.245,A -85,B 0,C 180,E1 -22615.111,E2 -22615.111} C_VEL
LIN {X 0,Y 178.463,Z 526.255,A -85,B 0,C 180,E1 -22620.794,E2 -22620.794} C_VEL
LIN {X 0,Y 178.485,Z 526.246,A -85,B 0,C 180,E1 -22624.218,E2 -22624.218} C_VEL
LIN {X 0,Y 178.392,Z 526.265,A -85,B 0,C 180,E1 -22629.075,E2 -22629.075} C_VEL
LIN {X 0,Y 178.397,Z 526.258,A -85,B 0,C 180,E1 -22632.045,E2 -22632.045} C_VEL
LIN {X 0,Y 178.395,Z 526.263,A -85,B 0,C 180,E1 -22635.164,E2 -22635.164} C_VEL
LIN {X 0,Y 178.405,Z 526.261,A -85,B 0,C 180,E1 -22638.459,E2 -22638.459} C_VEL
LIN {X 0,Y 178.425,Z 526.258,A -85,B 0,C 180,E1 -22643.783,E2 -22643.783} C_VEL
LIN {X 0,Y 178.489,Z 526.251,A -85,B 0,C 180,E1 -22646.546,E2 -22646.546} C_VEL
LIN {X 0,Y 178.525,Z 526.241,A -85,B 0,C 180,E1 -22650.006,E2 -22650.006} C_VEL
LIN {X 0,Y 178.522,Z 526.249,A -85,B 0,C 180,E1 -22654.885,E2 -22654.885} C_VEL
LIN {X 0,Y 178.624,Z 526.233,A -85,B 0,C 180,E1 -22660.784,E2 -22660.784} C_VEL
LIN {X 0,Y 178.661,Z 526.227,A -85,B 0,C 180,E1 -22666.347,E2 -22666.347} C_VEL
LIN {X 0,Y 178.908,Z 526.201,A -85,B 0,C 180,E1 -22670.959,E2 -22670.959} C_VEL
LIN {X 0,Y 179.15,Z 526.167,A -85,B 0,C 180,E1 -22677.751,E2 -22677.751} C_VEL
LIN {X 0,Y 179.366,Z 526.141,A -85,B 0,C 180,E1 -22679.999,E2 -22679.999} C_VEL
LIN {X 0,Y 178.849,Z 526.202,A -85,B 0,C 180,E1 -22684.507,E2 -22684.507} C_VEL
LIN {X 0,Y 178.905,Z 526.2,A -85,B 0,C 180,E1 -22689.04,E2 -22689.04} C_VEL
LIN {X 0,Y 178.652,Z 526.227,A -85,B 0,C 180,E1 -22693.652,E2 -22693.652} C_VEL
LIN {X 0,Y 178.62,Z 526.233,A -85,B 0,C 180,E1 -22699.213,E2 -22699.213} C_VEL
LIN {X 0,Y 178.515,Z 526.249,A -85,B 0,C 180,E1 -22705.111,E2 -22705.111} C_VEL
LIN {X 0,Y 178.46,Z 526.256,A -85,B 0,C 180,E1 -22710.794,E2 -22710.794} C_VEL
LIN {X 0,Y 178.553,Z 526.416,A -85,B 0,C 180,E1 -22714.04,E2 -22714.04} C_VEL
LIN {X 0,Y 179.627,Z 531.937,A -85,B 0,C 180,E1 -22718.756,E2 -22718.756} C_VEL
LIN {X 0,Y 181.005,Z 538.906,A -85,B 0,C 180,E1 -22724.338,E2 -22724.338} C_VEL
LIN {X 0,Y 182.324,Z 545.101,A -85,B 0,C 180,E1 -22729.058,E2 -22729.058} C_VEL
LIN {X 0,Y 182.401,Z 546.938,A -85,B 0,C 180,E1 -22730.408,E2 -22730.408} C_VEL
LIN {X 0,Y 181.001,Z 552.546,A -85,B 0,C 180,E1 -22734.379,E2 -22734.379} C_VEL
LIN {X 0,Y 179.962,Z 556.365,A -85,B 0,C 180,E1 -22737.083,E2 -22737.083} C_VEL
LIN {X 0,Y 180.863,Z 570.967,A -85,B 0,C 180,E1 -22738.451,E2 -22738.451} C_VEL
LIN {X 0,Y 181.431,Z 584.118,A -85,B 0,C 180,E1 -22740.084,E2 -22740.084} C_VEL
LIN {X 0,Y 181.669,Z 596.408,A -85,B 0,C 180,E1 -22742.027,E2 -22742.027} C_VEL
LIN {X 0,Y 181.645,Z 607.804,A -85,B 0,C 180,E1 -22744.244,E2 -22744.244} C_VEL
LIN {X 0,Y 181.445,Z 618.921,A -85,B 0,C 180,E1 -22746.91,E2 -22746.91} C_VEL
LIN {X 0,Y 181.058,Z 628.01,A -85,B 0,C 180,E1 -22749.553,E2 -22749.553} C_VEL
LIN {X 0,Y 179.659,Z 635.932,A -85,B 0,C 180,E1 -22752.352,E2 -22752.352} C_VEL
LIN {X 0,Y 178.462,Z 643.695,A -85,B 0,C 180,E1 -22755.752,E2 -22755.752} C_VEL
LIN {X 0,Y 178.038,Z 648.96,A -85,B 0,C 180,E1 -22758.617,E2 -22758.617} C_VEL
LIN {X 0,Y 178.014,Z 654.054,A -85,B 0,C 180,E1 -22762.058,E2 -22762.058} C_VEL
LIN {X 0,Y 178.459,Z 657.914,A -85,B 0,C 180,E1 -22765.483,E2 -22765.483} C_VEL
LIN {X 0,Y 178.828,Z 659.808,A -85,B 0,C 180,E1 -22767.748,E2 -22767.748} C_VEL
LIN {X 0,Y 179.249,Z 661.226,A -85,B 0,C 180,E1 -22770,E2 -22770} C_VEL
LIN {X 0,Y 178.584,Z 661.985,A -85,B 0,C 180,E1 -22772.256,E2 -22772.256} C_VEL
LIN {X 0,Y 177.964,Z 662.327,A -85,B 0,C 180,E1 -22774.53,E2 -22774.53} C_VEL
LIN {X 0,Y 177.287,Z 661.896,A -85,B 0,C 180,E1 -22778.637,E2 -22778.637} C_VEL
LIN {X 0,Y 177.264,Z 660.957,A -85,B 0,C 180,E1 -22781.434,E2 -22781.434} C_VEL
LIN {X 0,Y 178.264,Z 658.243,A -85,B 0,C 180,E1 -22786.02,E2 -22786.02} C_VEL
LIN {X 0,Y 179.217,Z 656.315,A -85,B 0,C 180,E1 -22788.301,E2 -22788.301} C_VEL
LIN {X 0,Y 179.609,Z 654.53,A -85,B 0,C 180,E1 -22790.093,E2 -22790.093} C_VEL
LIN {X 0,Y 178.946,Z 651.189,A -85,B 0,C 180,E1 -22793.077,E2 -22793.077} C_VEL
LIN {X 0,Y 178.817,Z 647.44,A -85,B 0,C 180,E1 -22796.008,E2 -22796.008} C_VEL
LIN {X 0,Y 180.011,Z 644.889,A -85,B 0,C 180,E1 -22797.662,E2 -22797.662} C_VEL
LIN {X 0,Y 183.983,Z 638.534,A -85,B 0,C 180,E1 -22801.044,E2 -22801.044} C_VEL
LIN {X 0,Y 188.746,Z 630.15,A -85,B 0,C 180,E1 -22804.607,E2 -22804.607} C_VEL
LIN {X 0,Y 192.067,Z 623.177,A -85,B 0,C 180,E1 -22807.14,E2 -22807.14} C_VEL
LIN {X 0,Y 195.682,Z 613.614,A -85,B 0,C 180,E1 -22810.277,E2 -22810.277} C_VEL
LIN {X 0,Y 198.225,Z 605.108,A -85,B 0,C 180,E1 -22812.911,E2 -22812.911} C_VEL
LIN {X 0,Y 200.702,Z 593.829,A -85,B 0,C 180,E1 -22816.341,E2 -22816.341} C_VEL
LIN {X 0,Y 201.346,Z 589.12,A -85,B 0,C 180,E1 -22817.888,E2 -22817.888} C_VEL
LIN {X 0,Y 200.598,Z 583.045,A -85,B 0,C 180,E1 -22820.903,E2 -22820.903} C_VEL
LIN {X 0,Y 199.402,Z 575.639,A -85,B 0,C 180,E1 -22825.673,E2 -22825.673} C_VEL
LIN {X 0,Y 198.766,Z 573.211,A -85,B 0,C 180,E1 -22828.06,E2 -22828.06} C_VEL
LIN {X 0,Y 198.329,Z 569.795,A -85,B 0,C 180,E1 -22832.57,E2 -22832.57} C_VEL
LIN {X 0,Y 198.917,Z 567.77,A -85,B 0,C 180,E1 -22837.13,E2 -22837.13} C_VEL
LIN {X 0,Y 199.486,Z 567.491,A -85,B 0,C 180,E1 -22839.372,E2 -22839.372} C_VEL
LIN {X 0,Y 200.912,Z 568.434,A -85,B 0,C 180,E1 -22843.75,E2 -22843.75} C_VEL
LIN {X 0,Y 201.677,Z 569.608,A -85,B 0,C 180,E1 -22845.882,E2 -22845.882} C_VEL
LIN {X 0,Y 202.181,Z 571.709,A -85,B 0,C 180,E1 -22847.962,E2 -22847.962} C_VEL
LIN {X 0,Y 202.921,Z 576.758,A -85,B 0,C 180,E1 -22852.037,E2 -22852.037} C_VEL
LIN {X 0,Y 203.297,Z 579.45,A -85,B 0,C 180,E1 -22854.048,E2 -22854.048} C_VEL
LIN {X 0,Y 203.245,Z 584.277,A -85,B 0,C 180,E1 -22857.027,E2 -22857.027} C_VEL
LIN {X 0,Y 202.775,Z 589.181,A -85,B 0,C 180,E1 -22860.001,E2 -22860.001} C_VEL
LIN {X 0,Y 202.109,Z 591.143,A -85,B 0,C 180,E1 -22860.997,E2 -22860.997} C_VEL
LIN {X 0,Y 196.4,Z 598.914,A -85,B 0,C 180,E1 -22864.105,E2 -22864.105} C_VEL
LIN {X 0,Y 191.315,Z 604.789,A -85,B 0,C 180,E1 -22867.314,E2 -22867.314} C_VEL
LIN {X 0,Y 186.229,Z 609.821,A -85,B 0,C 180,E1 -22871.124,E2 -22871.124} C_VEL
LIN {X 0,Y 181.943,Z 613.184,A -85,B 0,C 180,E1 -22875.05,E2 -22875.05} C_VEL
LIN {X 0,Y 178.446,Z 615.092,A -85,B 0,C 180,E1 -22879.049,E2 -22879.049} C_VEL
LIN {X 0,Y 175.519,Z 615.718,A -85,B 0,C 180,E1 -22883.605,E2 -22883.605} C_VEL
LIN {X 0,Y 173.819,Z 615.123,A -85,B 0,C 180,E1 -22887.185,E2 -22887.185} C_VEL
LIN {X 0,Y 172.599,Z 613.339,A -85,B 0,C 180,E1 -22891.229,E2 -22891.229} C_VEL
LIN {X 0,Y 172.06,Z 610.436,A -85,B 0,C 180,E1 -22895.221,E2 -22895.221} C_VEL
LIN {X 0,Y 172.15,Z 605.599,A -85,B 0,C 180,E1 -22899.834,E2 -22899.834} C_VEL
LIN {X 0,Y 172.872,Z 600.068,A -85,B 0,C 180,E1 -22903.72,E2 -22903.72} C_VEL
LIN {X 0,Y 174.088,Z 593.265,A -85,B 0,C 180,E1 -22907.458,E2 -22907.458} C_VEL
LIN {X 0,Y 175.487,Z 586.175,A -85,B 0,C 180,E1 -22910.61,E2 -22910.61} C_VEL
LIN {X 0,Y 177.345,Z 577.074,A -85,B 0,C 180,E1 -22913.906,E2 -22913.906} C_VEL
LIN {X 0,Y 179.313,Z 567.387,A -85,B 0,C 180,E1 -22916.72,E2 -22916.72} C_VEL
LIN {X 0,Y 180.776,Z 559.466,A -85,B 0,C 180,E1 -22918.648,E2 -22918.648} C_VEL
LIN {X 0,Y 178.343,Z 549.454,A -85,B 0,C 180,E1 -22921.128,E2 -22921.128} C_VEL
LIN {X 0,Y 175.299,Z 538.928,A -85,B 0,C 180,E1 -22923.433,E2 -22923.433} C_VEL
LIN {X 0,Y 171.469,Z 527.128,A -85,B 0,C 180,E1 -22925.725,E2 -22925.725} C_VEL
LIN {X 0,Y 171.58,Z 527.113,A -85,B 0,C 180,E1 -22930.871,E2 -22930.871} C_VEL
LIN {X 0,Y 171.573,Z 527.115,A -85,B 0,C 180,E1 -22935.772,E2 -22935.772} C_VEL
LIN {X 0,Y 171.848,Z 527.079,A -85,B 0,C 180,E1 -22940.585,E2 -22940.585} C_VEL
LIN {X 0,Y 171.812,Z 527.084,A -85,B 0,C 180,E1 -22945.307,E2 -22945.307} C_VEL
LIN {X 0,Y 172.33,Z 527.018,A -85,B 0,C 180,E1 -22950,E2 -22950} C_VEL
LIN {X 0,Y 171.807,Z 527.083,A -85,B 0,C 180,E1 -22954.692,E2 -22954.692} C_VEL
LIN {X 0,Y 171.847,Z 527.076,A -85,B 0,C 180,E1 -22959.415,E2 -22959.415} C_VEL
LIN {X 0,Y 171.573,Z 527.111,A -85,B 0,C 180,E1 -22964.227,E2 -22964.227} C_VEL
LIN {X 0,Y 171.543,Z 527.116,A -85,B 0,C 180,E1 -22969.557,E2 -22969.557} C_VEL
LIN {X 0,Y 171.447,Z 527.124,A -85,B 0,C 180,E1 -22975.598,E2 -22975.598} C_VEL
LIN {X 0,Y 171.42,Z 527.131,A -85,B 0,C 180,E1 -22980.572,E2 -22980.572} C_VEL
LIN {X 0,Y 171.394,Z 527.131,A -85,B 0,C 180,E1 -22985.034,E2 -22985.034} C_VEL
LIN {X 0,Y 171.347,Z 527.141,A -85,B 0,C 180,E1 -22988.801,E2 -22988.801} C_VEL
LIN {X 0,Y 171.321,Z 527.14,A -85,B 0,C 180,E1 -22994.217,E2 -22994.217} C_VEL
LIN {X 0,Y 171.337,Z 527.143,A -85,B 0,C 180,E1 -22998.981,E2 -22998.981} C_VEL
LIN {X 0,Y 171.389,Z 527.13,A -85,B 0,C 180,E1 -23002.04,E2 -23002.04} C_VEL
LIN {X 0,Y 171.4,Z 527.136,A -85,B 0,C 180,E1 -23005.092,E2 -23005.092} C_VEL
LIN {X 0,Y 171.451,Z 527.122,A -85,B 0,C 180,E1 -23010.534,E2 -23010.534} C_VEL
LIN {X 0,Y 171.447,Z 527.127,A -85,B 0,C 180,E1 -23015.799,E2 -23015.799} C_VEL
LIN {X 0,Y 171.58,Z 527.111,A -85,B 0,C 180,E1 -23020.871,E2 -23020.871} C_VEL
LIN {X 0,Y 171.578,Z 527.108,A -85,B 0,C 180,E1 -23025.772,E2 -23025.772} C_VEL
LIN {X 0,Y 171.846,Z 527.078,A -85,B 0,C 180,E1 -23030.584,E2 -23030.584} C_VEL
LIN {X 0,Y 171.808,Z 527.078,A -85,B 0,C 180,E1 -23035.307,E2 -23035.307} C_VEL
LIN {X 0,Y 172.329,Z 527.018,A -85,B 0,C 180,E1 -23039.999,E2 -23039.999} C_VEL
LIN {X 0,Y 171.798,Z 527.081,A -85,B 0,C 180,E1 -23044.692,E2 -23044.692} C_VEL
LIN {X 0,Y 171.844,Z 527.078,A -85,B 0,C 180,E1 -23049.415,E2 -23049.415} C_VEL
LIN {X 0,Y 171.569,Z 527.109,A -85,B 0,C 180,E1 -23054.227,E2 -23054.227} C_VEL
LIN {X 0,Y 171.539,Z 527.114,A -85,B 0,C 180,E1 -23059.556,E2 -23059.556} C_VEL
LIN {X 0,Y 171.444,Z 527.128,A -85,B 0,C 180,E1 -23065.598,E2 -23065.598} C_VEL
LIN {X 0,Y 171.417,Z 527.132,A -85,B 0,C 180,E1 -23070.572,E2 -23070.572} C_VEL
LIN {X 0,Y 171.496,Z 527.215,A -85,B 0,C 180,E1 -23073.589,E2 -23073.589} C_VEL
LIN {X 0,Y 172.384,Z 531.834,A -85,B 0,C 180,E1 -23077.701,E2 -23077.701} C_VEL
LIN {X 0,Y 173.735,Z 538.697,A -85,B 0,C 180,E1 -23083.447,E2 -23083.447} C_VEL
LIN {X 0,Y 175.263,Z 545.785,A -85,B 0,C 180,E1 -23089.111,E2 -23089.111} C_VEL
LIN {X 0,Y 175.318,Z 547.083,A -85,B 0,C 180,E1 -23090.104,E2 -23090.104} C_VEL
LIN {X 0,Y 174.468,Z 550.788,A -85,B 0,C 180,E1 -23092.826,E2 -23092.826} C_VEL
LIN {X 0,Y 173.132,Z 555.557,A -85,B 0,C 180,E1 -23096.291,E2 -23096.291} C_VEL
LIN {X 0,Y 173.954,Z 569.764,A -85,B 0,C 180,E1 -23097.636,E2 -23097.636} C_VEL
LIN {X 0,Y 174.449,Z 582.439,A -85,B 0,C 180,E1 -23099.26,E2 -23099.26} C_VEL
LIN {X 0,Y 174.689,Z 596.111,A -85,B 0,C 180,E1 -23101.52,E2 -23101.52} C_VEL
LIN {X 0,Y 174.617,Z 608.264,A -85,B 0,C 180,E1 -23104.043,E2 -23104.043} C_VEL
LIN {X 0,Y 174.352,Z 619.151,A -85,B 0,C 180,E1 -23106.828,E2 -23106.828} C_VEL
LIN {X 0,Y 174.007,Z 627.211,A -85,B 0,C 180,E1 -23109.304,E2 -23109.304} C_VEL
LIN {X 0,Y 172.619,Z 635.101,A -85,B 0,C 180,E1 -23112.221,E2 -23112.221} C_VEL
LIN {X 0,Y 171.429,Z 642.817,A -85,B 0,C 180,E1 -23115.761,E2 -23115.761} C_VEL
LIN {X 0,Y 170.99,Z 648.976,A -85,B 0,C 180,E1 -23119.342,E2 -23119.342} C_VEL
LIN {X 0,Y 171.093,Z 653.805,A -85,B 0,C 180,E1 -23122.922,E2 -23122.922} C_VEL
LIN {X 0,Y 171.58,Z 657.414,A -85,B 0,C 180,E1 -23126.478,E2 -23126.478} C_VEL
LIN {X 0,Y 172.245,Z 659.879,A -85,B 0,C 180,E1 -23130,E2 -23130} C_VEL
LIN {X 0,Y 171.563,Z 660.692,A -85,B 0,C 180,E1 -23132.348,E2 -23132.348} C_VEL
LIN {X 0,Y 170.493,Z 661.107,A -85,B 0,C 180,E1 -23137.104,E2 -23137.104} C_VEL
LIN {X 0,Y 170.271,Z 659.986,A -85,B 0,C 180,E1 -23141.91,E2 -23141.91} C_VEL
LIN {X 0,Y 171.393,Z 657.431,A -85,B 0,C 180,E1 -23146.681,E2 -23146.681} C_VEL
LIN {X 0,Y 173.806,Z 653.449,A -85,B 0,C 180,E1 -23151.342,E2 -23151.342} C_VEL
LIN {X 0,Y 177.84,Z 647.89,A -85,B 0,C 180,E1 -23155.767,E2 -23155.767} C_VEL
LIN {X 0,Y 180.011,Z 644.889,A -85,B 0,C 180,E1 -23157.662,E2 -23157.662} C_VEL
LIN {X 0,Y 181.286,Z 642.225,A -85,B 0,C 180,E1 -23159.279,E2 -23159.279} C_VEL
LIN {X 0,Y 181.737,Z 637.71,A -85,B 0,C 180,E1 -23162.056,E2 -23162.056} C_VEL
LIN {X 0,Y 182.225,Z 632.799,A -85,B 0,C 180,E1 -23164.785,E2 -23164.785} C_VEL
LIN {X 0,Y 183.529,Z 629.505,A -85,B 0,C 180,E1 -23166.281,E2 -23166.281} C_VEL
LIN {X 0,Y 187.741,Z 620.939,A -85,B 0,C 180,E1 -23169.523,E2 -23169.523} C_VEL
LIN {X 0,Y 191.626,Z 611.29,A -85,B 0,C 180,E1 -23172.819,E2 -23172.819} C_VEL
LIN {X 0,Y 195.324,Z 598.874,A -85,B 0,C 180,E1 -23176.871,E2 -23176.871} C_VEL
LIN {X 0,Y 196.457,Z 593.51,A -85,B 0,C 180,E1 -23178.7,E2 -23178.7} C_VEL
LIN {X 0,Y 195.928,Z 586.707,A -85,B 0,C 180,E1 -23182.426,E2 -23182.426} C_VEL
LIN {X 0,Y 195.456,Z 581.817,A -85,B 0,C 180,E1 -23185.794,E2 -23185.794} C_VEL
LIN {X 0,Y 195.035,Z 579.262,A -85,B 0,C 180,E1 -23188.208,E2 -23188.208} C_VEL
LIN {X 0,Y 194.679,Z 576.35,A -85,B 0,C 180,E1 -23192.011,E2 -23192.011} C_VEL
LIN {X 0,Y 195.166,Z 574.081,A -85,B 0,C 180,E1 -23196.665,E2 -23196.665} C_VEL
LIN {X 0,Y 195.668,Z 573.585,A -85,B 0,C 180,E1 -23199.048,E2 -23199.048} C_VEL
LIN {X 0,Y 196.845,Z 574.268,A -85,B 0,C 180,E1 -23203.404,E2 -23203.404} C_VEL
LIN {X 0,Y 197.499,Z 575.272,A -85,B 0,C 180,E1 -23205.577,E2 -23205.577} C_VEL
LIN {X 0,Y 197.842,Z 578.315,A -85,B 0,C 180,E1 -23208.734,E2 -23208.734} C_VEL
LIN {X 0,Y 198.169,Z 583.662,A -85,B 0,C 180,E1 -23213.226,E2 -23213.226} C_VEL
LIN {X 0,Y 197.875,Z 587.525,A -85,B 0,C 180,E1 -23215.927,E2 -23215.927} C_VEL
LIN {X 0,Y 197.128,Z 592.29,A -85,B 0,C 180,E1 -23219.081,E2 -23219.081} C_VEL
LIN {X 0,Y 196.417,Z 593.98,A -85,B 0,C 180,E1 -23220.001,E2 -23220.001} C_VEL
LIN {X 0,Y 190.698,Z 601.062,A -85,B 0,C 180,E1 -23223.021,E2 -23223.021} C_VEL
LIN {X 0,Y 185.019,Z 607.106,A -85,B 0,C 180,E1 -23226.544,E2 -23226.544} C_VEL
LIN {X 0,Y 180.281,Z 611.293,A -85,B 0,C 180,E1 -23229.951,E2 -23229.951} C_VEL
LIN {X 0,Y 175.858,Z 614.451,A -85,B 0,C 180,E1 -23233.874,E2 -23233.874} C_VEL
LIN {X 0,Y 173.401,Z 615.792,A -85,B 0,C 180,E1 -23236.483,E2 -23236.483} C_VEL
LIN {X 0,Y 171.175,Z 616.61,A -85,B 0,C 180,E1 -23239.208,E2 -23239.208} C_VEL
LIN {X 0,Y 168.502,Z 616.798,A -85,B 0,C 180,E1 -23243.422,E2 -23243.422} C_VEL
LIN {X 0,Y 166.56,Z 615.802,A -85,B 0,C 180,E1 -23247.656,E2 -23247.656} C_VEL
LIN {X 0,Y 165.425,Z 613.683,A -85,B 0,C 180,E1 -23251.821,E2 -23251.821} C_VEL
LIN {X 0,Y 164.932,Z 609.796,A -85,B 0,C 180,E1 -23256.625,E2 -23256.625} C_VEL
LIN {X 0,Y 165.264,Z 604.439,A -85,B 0,C 180,E1 -23261.288,E2 -23261.288} C_VEL
LIN {X 0,Y 166.057,Z 599.184,A -85,B 0,C 180,E1 -23264.807,E2 -23264.807} C_VEL
LIN {X 0,Y 167.256,Z 592.818,A -85,B 0,C 180,E1 -23268.266,E2 -23268.266} C_VEL
LIN {X 0,Y 168.814,Z 585.116,A -85,B 0,C 180,E1 -23271.654,E2 -23271.654} C_VEL
LIN {X 0,Y 170.991,Z 574.774,A -85,B 0,C 180,E1 -23275.29,E2 -23275.29} C_VEL
LIN {X 0,Y 173.119,Z 564.574,A -85,B 0,C 180,E1 -23278.146,E2 -23278.146} C_VEL
LIN {X 0,Y 173.786,Z 560.313,A -85,B 0,C 180,E1 -23279.19,E2 -23279.19} C_VEL
LIN {X 0,Y 171.206,Z 549.92,A -85,B 0,C 180,E1 -23281.875,E2 -23281.875} C_VEL
LIN {X 0,Y 168.104,Z 539.203,A -85,B 0,C 180,E1 -23284.32,E2 -23284.32} C_VEL
LIN {X 0,Y 164.368,Z 528.011,A -85,B 0,C 180,E1 -23286.618,E2 -23286.618} C_VEL
LIN {X 0,Y 164.484,Z 527.997,A -85,B 0,C 180,E1 -23290.055,E2 -23290.055} C_VEL
LIN {X 0,Y 164.503,Z 527.996,A -85,B 0,C 180,E1 -23295.147,E2 -23295.147} C_VEL
LIN {X 0,Y 164.769,Z 527.961,A -85,B 0,C 180,E1 -23300.176,E2 -23300.176} C_VEL
LIN {X 0,Y 164.829,Z 527.952,A -85,B 0,C 180,E1 -23302.651,E2 -23302.651} C_VEL
LIN {X 0,Y 165.048,Z 527.926,A -85,B 0,C 180,E1 -23307.559,E2 -23307.559} C_VEL
LIN {X 0,Y 165.293,Z 527.894,A -85,B 0,C 180,E1 -23310,E2 -23310} C_VEL
LIN {X 0,Y 164.756,Z 527.962,A -85,B 0,C 180,E1 -23314.894,E2 -23314.894} C_VEL
LIN {X 0,Y 164.826,Z 527.95,A -85,B 0,C 180,E1 -23317.349,E2 -23317.349} C_VEL
LIN {X 0,Y 164.705,Z 527.967,A -85,B 0,C 180,E1 -23321.059,E2 -23321.059} C_VEL
LIN {X 0,Y 164.482,Z 527.992,A -85,B 0,C 180,E1 -23327.403,E2 -23327.403} C_VEL
LIN {X 0,Y 164.476,Z 527.995,A -85,B 0,C 180,E1 -23329.989,E2 -23329.989} C_VEL
LIN {X 0,Y 164.373,Z 528.004,A -85,B 0,C 180,E1 -23336.117,E2 -23336.117} C_VEL
LIN {X 0,Y 164.36,Z 528.012,A -85,B 0,C 180,E1 -23341.217,E2 -23341.217} C_VEL
LIN {X 0,Y 164.283,Z 528.019,A -85,B 0,C 180,E1 -23346.792,E2 -23346.792} C_VEL
LIN {X 0,Y 164.289,Z 528.019,A -85,B 0,C 180,E1 -23349.917,E2 -23349.917} C_VEL
LIN {X 0,Y 164.281,Z 528.017,A -85,B 0,C 180,E1 -23353.341,E2 -23353.341} C_VEL
LIN {X 0,Y 164.265,Z 528.023,A -85,B 0,C 180,E1 -23356.798,E2 -23356.798} C_VEL
LIN {X 0,Y 164.297,Z 528.016,A -85,B 0,C 180,E1 -23360.351,E2 -23360.351} C_VEL
LIN {X 0,Y 164.332,Z 528.013,A -85,B 0,C 180,E1 -23364.348,E2 -23364.348} C_VEL
LIN {X 0,Y 164.393,Z 528.003,A -85,B 0,C 180,E1 -23369.134,E2 -23369.134} C_VEL
LIN {X 0,Y 164.409,Z 528.006,A -85,B 0,C 180,E1 -23374.692,E2 -23374.692} C_VEL
LIN {X 0,Y 164.486,Z 527.992,A -85,B 0,C 180,E1 -23380.051,E2 -23380.051} C_VEL
LIN {X 0,Y 164.526,Z 527.989,A -85,B 0,C 180,E1 -23385.149,E2 -23385.149} C_VEL
LIN {X 0,Y 164.767,Z 527.959,A -85,B 0,C 180,E1 -23390.176,E2 -23390.176} C_VEL
LIN {X 0,Y 164.826,Z 527.954,A -85,B 0,C 180,E1 -23392.65,E2 -23392.65} C_VEL
LIN {X 0,Y 165.045,Z 527.924,A -85,B 0,C 180,E1 -23397.559,E2 -23397.559} C_VEL
LIN {X 0,Y 165.291,Z 527.894,A -85,B 0,C 180,E1 -23399.999,E2 -23399.999} C_VEL
LIN {X 0,Y 164.747,Z 527.959,A -85,B 0,C 180,E1 -23404.894,E2 -23404.894} C_VEL
LIN {X 0,Y 164.822,Z 527.954,A -85,B 0,C 180,E1 -23407.349,E2 -23407.349} C_VEL
LIN {X 0,Y 164.702,Z 527.966,A -85,B 0,C 180,E1 -23411.059,E2 -23411.059} C_VEL
LIN {X 0,Y 164.478,Z 527.996,A -85,B 0,C 180,E1 -23417.403,E2 -23417.403} C_VEL
LIN {X 0,Y 164.473,Z 527.994,A -85,B 0,C 180,E1 -23419.989,E2 -23419.989} C_VEL
LIN {X 0,Y 164.37,Z 528.009,A -85,B 0,C 180,E1 -23426.117,E2 -23426.117} C_VEL
LIN {X 0,Y 164.406,Z 528.012,A -85,B 0,C 180,E1 -23432.362,E2 -23432.362} C_VEL
LIN {X 0,Y 164.45,Z 528.142,A -85,B 0,C 180,E1 -23433.223,E2 -23433.223} C_VEL
LIN {X 0,Y 165.451,Z 533.339,A -85,B 0,C 180,E1 -23438.019,E2 -23438.019} C_VEL
LIN {X 0,Y 166.688,Z 539.457,A -85,B 0,C 180,E1 -23443.371,E2 -23443.371} C_VEL
LIN {X 0,Y 168.122,Z 545.973,A -85,B 0,C 180,E1 -23448.803,E2 -23448.803} C_VEL
LIN {X 0,Y 168.231,Z 547.514,A -85,B 0,C 180,E1 -23450.026,E2 -23450.026} C_VEL
LIN {X 0,Y 166.885,Z 552.508,A -85,B 0,C 180,E1 -23453.873,E2 -23453.873} C_VEL
LIN {X 0,Y 166.336,Z 554.487,A -85,B 0,C 180,E1 -23455.406,E2 -23455.406} C_VEL
LIN {X 0,Y 167.089,Z 569.097,A -85,B 0,C 180,E1 -23456.852,E2 -23456.852} C_VEL
LIN {X 0,Y 167.546,Z 582.272,A -85,B 0,C 180,E1 -23458.631,E2 -23458.631} C_VEL
LIN {X 0,Y 167.711,Z 595.827,A -85,B 0,C 180,E1 -23460.983,E2 -23460.983} C_VEL
LIN {X 0,Y 167.584,Z 607.532,A -85,B 0,C 180,E1 -23463.54,E2 -23463.54} C_VEL
LIN {X 0,Y 167.286,Z 618.93,A -85,B 0,C 180,E1 -23466.609,E2 -23466.609} C_VEL
LIN {X 0,Y 166.948,Z 626.404,A -85,B 0,C 180,E1 -23469.034,E2 -23469.034} C_VEL
LIN {X 0,Y 165.892,Z 632.832,A -85,B 0,C 180,E1 -23471.474,E2 -23471.474} C_VEL
LIN {X 0,Y 164.48,Z 640.736,A -85,B 0,C 180,E1 -23475.145,E2 -23475.145} C_VEL
LIN {X 0,Y 164.006,Z 647.134,A -85,B 0,C 180,E1 -23478.882,E2 -23478.882} C_VEL
LIN {X 0,Y 164.054,Z 652.132,A -85,B 0,C 180,E1 -23482.616,E2 -23482.616} C_VEL
LIN {X 0,Y 164.553,Z 655.895,A -85,B 0,C 180,E1 -23486.327,E2 -23486.327} C_VEL
LIN {X 0,Y 165.237,Z 658.493,A -85,B 0,C 180,E1 -23490,E2 -23490} C_VEL
LIN {X 0,Y 164.535,Z 659.379,A -85,B 0,C 180,E1 -23492.448,E2 -23492.448} C_VEL
LIN {X 0,Y 163.429,Z 659.923,A -85,B 0,C 180,E1 -23497.413,E2 -23497.413} C_VEL
LIN {X 0,Y 163.269,Z 658.988,A -85,B 0,C 180,E1 -23502.429,E2 -23502.429} C_VEL
LIN {X 0,Y 164.552,Z 656.629,A -85,B 0,C 180,E1 -23507.396,E2 -23507.396} C_VEL
LIN {X 0,Y 167.354,Z 652.572,A -85,B 0,C 180,E1 -23512.5,E2 -23512.5} C_VEL
LIN {X 0,Y 171.433,Z 647.575,A -85,B 0,C 180,E1 -23516.805,E2 -23516.805} C_VEL
LIN {X 0,Y 175.316,Z 642.503,A -85,B 0,C 180,E1 -23520.073,E2 -23520.073} C_VEL
LIN {X 0,Y 179.973,Z 635.318,A -85,B 0,C 180,E1 -23523.812,E2 -23523.812} C_VEL
LIN {X 0,Y 183.529,Z 629.505,A -85,B 0,C 180,E1 -23526.281,E2 -23526.281} C_VEL
LIN {X 0,Y 184.811,Z 626.195,A -85,B 0,C 180,E1 -23527.746,E2 -23527.746} C_VEL
LIN {X 0,Y 185.273,Z 621.045,A -85,B 0,C 180,E1 -23530.364,E2 -23530.364} C_VEL
LIN {X 0,Y 185.802,Z 614.6,A -85,B 0,C 180,E1 -23533.495,E2 -23533.495} C_VEL
LIN {X 0,Y 186.564,Z 612.179,A -85,B 0,C 180,E1 -23534.444,E2 -23534.444} C_VEL
LIN {X 0,Y 189.956,Z 602.799,A -85,B 0,C 180,E1 -23537.729,E2 -23537.729} C_VEL
LIN {X 0,Y 191.283,Z 598.508,A -85,B 0,C 180,E1 -23539.251,E2 -23539.251} C_VEL
LIN {X 0,Y 191.515,Z 597.223,A -85,B 0,C 180,E1 -23539.795,E2 -23539.795} C_VEL
LIN {X 0,Y 191.424,Z 592.169,A -85,B 0,C 180,E1 -23542.715,E2 -23542.715} C_VEL
LIN {X 0,Y 191.131,Z 586.961,A -85,B 0,C 180,E1 -23546.526,E2 -23546.526} C_VEL
LIN {X 0,Y 190.883,Z 584.609,A -85,B 0,C 180,E1 -23548.972,E2 -23548.972} C_VEL
LIN {X 0,Y 190.774,Z 581.359,A -85,B 0,C 180,E1 -23553.764,E2 -23553.764} C_VEL
LIN {X 0,Y 191.221,Z 579.997,A -85,B 0,C 180,E1 -23556.757,E2 -23556.757} C_VEL
LIN {X 0,Y 191.521,Z 579.565,A -85,B 0,C 180,E1 -23558.472,E2 -23558.472} C_VEL
LIN {X 0,Y 192.524,Z 579.918,A -85,B 0,C 180,E1 -23563.021,E2 -23563.021} C_VEL
LIN {X 0,Y 193.089,Z 580.749,A -85,B 0,C 180,E1 -23565.24,E2 -23565.24} C_VEL
LIN {X 0,Y 193.125,Z 582.519,A -85,B 0,C 180,E1 -23567.389,E2 -23567.389} C_VEL
LIN {X 0,Y 192.982,Z 586.939,A -85,B 0,C 180,E1 -23571.624,E2 -23571.624} C_VEL
LIN {X 0,Y 192.832,Z 589.426,A -85,B 0,C 180,E1 -23573.723,E2 -23573.723} C_VEL
LIN {X 0,Y 191.572,Z 595.106,A -85,B 0,C 180,E1 -23577.898,E2 -23577.898} C_VEL
LIN {X 0,Y 190.867,Z 596.706,A -85,B 0,C 180,E1 -23578.909,E2 -23578.909} C_VEL
LIN {X 0,Y 184.568,Z 603.815,A -85,B 0,C 180,E1 -23582.183,E2 -23582.183} C_VEL
LIN {X 0,Y 178.867,Z 609.241,A -85,B 0,C 180,E1 -23585.638,E2 -23585.638} C_VEL
LIN {X 0,Y 173.665,Z 613.328,A -85,B 0,C 180,E1 -23589.316,E2 -23589.316} C_VEL
LIN {X 0,Y 170.684,Z 615.31,A -85,B 0,C 180,E1 -23591.882,E2 -23591.882} C_VEL
LIN {X 0,Y 167.405,Z 616.952,A -85,B 0,C 180,E1 -23595.073,E2 -23595.073} C_VEL
LIN {X 0,Y 163.879,Z 617.999,A -85,B 0,C 180,E1 -23599.354,E2 -23599.354} C_VEL
LIN {X 0,Y 161.217,Z 617.779,A -85,B 0,C 180,E1 -23603.727,E2 -23603.727} C_VEL
LIN {X 0,Y 159.335,Z 616.399,A -85,B 0,C 180,E1 -23608.094,E2 -23608.094} C_VEL
LIN {X 0,Y 158.073,Z 612.928,A -85,B 0,C 180,E1 -23613.786,E2 -23613.786} C_VEL
LIN {X 0,Y 157.885,Z 608.434,A -85,B 0,C 180,E1 -23618.55,E2 -23618.55} C_VEL
LIN {X 0,Y 158.398,Z 603.401,A -85,B 0,C 180,E1 -23622.575,E2 -23622.575} C_VEL
LIN {X 0,Y 159.516,Z 596.976,A -85,B 0,C 180,E1 -23626.634,E2 -23626.634} C_VEL
LIN {X 0,Y 161.225,Z 588.515,A -85,B 0,C 180,E1 -23630.829,E2 -23630.829} C_VEL
LIN {X 0,Y 163.045,Z 580.002,A -85,B 0,C 180,E1 -23634.219,E2 -23634.219} C_VEL
LIN {X 0,Y 165.323,Z 569.615,A -85,B 0,C 180,E1 -23637.537,E2 -23637.537} C_VEL
LIN {X 0,Y 166.883,Z 561.642,A -85,B 0,C 180,E1 -23639.644,E2 -23639.644} C_VEL
LIN {X 0,Y 164.454,Z 551.805,A -85,B 0,C 180,E1 -23642.306,E2 -23642.306} C_VEL
LIN {X 0,Y 161.383,Z 541.055,A -85,B 0,C 180,E1 -23644.874,E2 -23644.874} C_VEL
LIN {X 0,Y 157.335,Z 528.888,A -85,B 0,C 180,E1 -23647.512,E2 -23647.512} C_VEL
LIN {X 0,Y 157.409,Z 528.879,A -85,B 0,C 180,E1 -23651.787,E2 -23651.787} C_VEL
LIN {X 0,Y 157.527,Z 528.865,A -85,B 0,C 180,E1 -23657.11,E2 -23657.11} C_VEL
LIN {X 0,Y 157.692,Z 528.844,A -85,B 0,C 180,E1 -23659.73,E2 -23659.73} C_VEL
LIN {X 0,Y 157.766,Z 528.832,A -85,B 0,C 180,E1 -23662.32,E2 -23662.32} C_VEL
LIN {X 0,Y 158.256,Z 528.771,A -85,B 0,C 180,E1 -23670,E2 -23670} C_VEL
LIN {X 0,Y 157.764,Z 528.828,A -85,B 0,C 180,E1 -23677.68,E2 -23677.68} C_VEL
LIN {X 0,Y 157.636,Z 528.848,A -85,B 0,C 180,E1 -23681.229,E2 -23681.229} C_VEL
LIN {X 0,Y 157.441,Z 528.87,A -85,B 0,C 180,E1 -23685.535,E2 -23685.535} C_VEL
LIN {X 0,Y 157.37,Z 528.882,A -85,B 0,C 180,E1 -23690.933,E2 -23690.933} C_VEL
LIN {X 0,Y 157.312,Z 528.884,A -85,B 0,C 180,E1 -23696.68,E2 -23696.68} C_VEL
LIN {X 0,Y 157.27,Z 528.892,A -85,B 0,C 180,E1 -23702.428,E2 -23702.428} C_VEL
LIN {X 0,Y 157.261,Z 528.893,A -85,B 0,C 180,E1 -23706.444,E2 -23706.444} C_VEL
LIN {X 0,Y 157.193,Z 528.899,A -85,B 0,C 180,E1 -23712.116,E2 -23712.116} C_VEL
LIN {X 0,Y 157.195,Z 528.903,A -85,B 0,C 180,E1 -23717.883,E2 -23717.883} C_VEL
LIN {X 0,Y 157.27,Z 528.893,A -85,B 0,C 180,E1 -23723.55,E2 -23723.55} C_VEL
LIN {X 0,Y 157.296,Z 528.889,A -85,B 0,C 180,E1 -23728.095,E2 -23728.095} C_VEL
LIN {X 0,Y 157.317,Z 528.889,A -85,B 0,C 180,E1 -23733.464,E2 -23733.464} C_VEL
LIN {X 0,Y 157.394,Z 528.875,A -85,B 0,C 180,E1 -23739.668,E2 -23739.668} C_VEL
LIN {X 0,Y 157.456,Z 528.871,A -85,B 0,C 180,E1 -23744.465,E2 -23744.465} C_VEL
LIN {X 0,Y 157.689,Z 528.841,A -85,B 0,C 180,E1 -23749.73,E2 -23749.73} C_VEL
LIN {X 0,Y 157.764,Z 528.832,A -85,B 0,C 180,E1 -23752.319,E2 -23752.319} C_VEL
LIN {X 0,Y 158.254,Z 528.771,A -85,B 0,C 180,E1 -23759.999,E2 -23759.999} C_VEL
LIN {X 0,Y 157.76,Z 528.833,A -85,B 0,C 180,E1 -23767.68,E2 -23767.68} C_VEL
LIN {X 0,Y 157.633,Z 528.846,A -85,B 0,C 180,E1 -23771.229,E2 -23771.229} C_VEL
LIN {X 0,Y 157.437,Z 528.872,A -85,B 0,C 180,E1 -23775.535,E2 -23775.535} C_VEL
LIN {X 0,Y 157.366,Z 528.878,A -85,B 0,C 180,E1 -23780.933,E2 -23780.933} C_VEL
LIN {X 0,Y 157.309,Z 528.891,A -85,B 0,C 180,E1 -23786.68,E2 -23786.68} C_VEL
LIN {X 0,Y 157.381,Z 528.96,A -85,B 0,C 180,E1 -23792.782,E2 -23792.782} C_VEL
LIN {X 0,Y 158.505,Z 534.782,A -85,B 0,C 180,E1 -23798.37,E2 -23798.37} C_VEL
LIN {X 0,Y 159.569,Z 539.926,A -85,B 0,C 180,E1 -23803.052,E2 -23803.052} C_VEL
LIN {X 0,Y 161.065,Z 546.918,A -85,B 0,C 180,E1 -23809.117,E2 -23809.117} C_VEL
LIN {X 0,Y 160.928,Z 548.873,A -85,B 0,C 180,E1 -23810.712,E2 -23810.712} C_VEL
LIN {X 0,Y 159.52,Z 553.528,A -85,B 0,C 180,E1 -23814.479,E2 -23814.479} C_VEL
LIN {X 0,Y 160.158,Z 567.026,A -85,B 0,C 180,E1 -23815.855,E2 -23815.855} C_VEL
LIN {X 0,Y 160.583,Z 579.407,A -85,B 0,C 180,E1 -23817.548,E2 -23817.548} C_VEL
LIN {X 0,Y 160.668,Z 591.998,A -85,B 0,C 180,E1 -23819.745,E2 -23819.745} C_VEL
LIN {X 0,Y 160.555,Z 603.717,A -85,B 0,C 180,E1 -23822.284,E2 -23822.284} C_VEL
LIN {X 0,Y 160.369,Z 614.201,A -85,B 0,C 180,E1 -23825.052,E2 -23825.052} C_VEL
LIN {X 0,Y 160.002,Z 623.9,A -85,B 0,C 180,E1 -23828.169,E2 -23828.169} C_VEL
LIN {X 0,Y 159.473,Z 628.849,A -85,B 0,C 180,E1 -23830.029,E2 -23830.029} C_VEL
LIN {X 0,Y 157.844,Z 637.343,A -85,B 0,C 180,E1 -23833.843,E2 -23833.843} C_VEL
LIN {X 0,Y 157.1,Z 644.164,A -85,B 0,C 180,E1 -23837.732,E2 -23837.732} C_VEL
LIN {X 0,Y 157.056,Z 650.35,A -85,B 0,C 180,E1 -23842.285,E2 -23842.285} C_VEL
LIN {X 0,Y 157.553,Z 654.293,A -85,B 0,C 180,E1 -23846.164,E2 -23846.164} C_VEL
LIN {X 0,Y 158.248,Z 657.045,A -85,B 0,C 180,E1 -23850,E2 -23850} C_VEL
LIN {X 0,Y 157.502,Z 658.037,A -85,B 0,C 180,E1 -23852.558,E2 -23852.558} C_VEL
LIN {X 0,Y 156.798,Z 658.582,A -85,B 0,C 180,E1 -23855.144,E2 -23855.144} C_VEL
LIN {X 0,Y 156.149,Z 658.511,A -85,B 0,C 180,E1 -23860.372,E2 -23860.372} C_VEL
LIN {X 0,Y 156.847,Z 657.046,A -85,B 0,C 180,E1 -23865.596,E2 -23865.596} C_VEL
LIN {X 0,Y 158.938,Z 654.202,A -85,B 0,C 180,E1 -23870.717,E2 -23870.717} C_VEL
LIN {X 0,Y 161.607,Z 651.119,A -85,B 0,C 180,E1 -23874.403,E2 -23874.403} C_VEL
LIN {X 0,Y 165.103,Z 647.177,A -85,B 0,C 180,E1 -23877.921,E2 -23877.921} C_VEL
LIN {X 0,Y 169.131,Z 642.351,A -85,B 0,C 180,E1 -23881.294,E2 -23881.294} C_VEL
LIN {X 0,Y 174.097,Z 635.467,A -85,B 0,C 180,E1 -23885.118,E2 -23885.118} C_VEL
LIN {X 0,Y 178.488,Z 628.74,A -85,B 0,C 180,E1 -23888.14,E2 -23888.14} C_VEL
LIN {X 0,Y 182.967,Z 620.321,A -85,B 0,C 180,E1 -23891.499,E2 -23891.499} C_VEL
LIN {X 0,Y 186.564,Z 612.179,A -85,B 0,C 180,E1 -23894.444,E2 -23894.444} C_VEL
LIN {X 0,Y 187.537,Z 608.672,A -85,B 0,C 180,E1 -23895.882,E2 -23895.882} C_VEL
LIN {X 0,Y 187.725,Z 605.594,A -85,B 0,C 180,E1 -23897.449,E2 -23897.449} C_VEL
LIN {X 0,Y 187.57,Z 603.775,A -85,B 0,C 180,E1 -23898.535,E2 -23898.535} C_VEL
LIN {X 0,Y 186.562,Z 597.343,A -85,B 0,C 180,E1 -23903.127,E2 -23903.127} C_VEL
LIN {X 0,Y 186.617,Z 592.322,A -85,B 0,C 180,E1 -23906.922,E2 -23906.922} C_VEL
LIN {X 0,Y 186.64,Z 590.991,A -85,B 0,C 180,E1 -23908.186,E2 -23908.186} C_VEL
LIN {X 0,Y 186.47,Z 587.497,A -85,B 0,C 180,E1 -23913.111,E2 -23913.111} C_VEL
LIN {X 0,Y 187.152,Z 585.404,A -85,B 0,C 180,E1 -23917.944,E2 -23917.944} C_VEL
LIN {X 0,Y 187.532,Z 585.211,A -85,B 0,C 180,E1 -23920.289,E2 -23920.289} C_VEL
LIN {X 0,Y 187.998,Z 585.388,A -85,B 0,C 180,E1 -23922.599,E2 -23922.599} C_VEL
LIN {X 0,Y 188.443,Z 586.049,A -85,B 0,C 180,E1 -23924.867,E2 -23924.867} C_VEL
LIN {X 0,Y 188.306,Z 587.639,A -85,B 0,C 180,E1 -23927.06,E2 -23927.06} C_VEL
LIN {X 0,Y 187.912,Z 590.658,A -85,B 0,C 180,E1 -23930.311,E2 -23930.311} C_VEL
LIN {X 0,Y 187.296,Z 594.095,A -85,B 0,C 180,E1 -23933.537,E2 -23933.537} C_VEL
LIN {X 0,Y 186.044,Z 598.021,A -85,B 0,C 180,E1 -23936.752,E2 -23936.752} C_VEL
LIN {X 0,Y 185.237,Z 599.575,A -85,B 0,C 180,E1 -23937.826,E2 -23937.826} C_VEL
LIN {X 0,Y 178.718,Z 606.249,A -85,B 0,C 180,E1 -23941.127,E2 -23941.127} C_VEL
LIN {X 0,Y 172.742,Z 611.379,A -85,B 0,C 180,E1 -23944.668,E2 -23944.668} C_VEL
LIN {X 0,Y 167.297,Z 615.19,A -85,B 0,C 180,E1 -23948.456,E2 -23948.456} C_VEL
LIN {X 0,Y 162.668,Z 617.688,A -85,B 0,C 180,E1 -23952.476,E2 -23952.476} C_VEL
LIN {X 0,Y 159.916,Z 618.69,A -85,B 0,C 180,E1 -23955.29,E2 -23955.29} C_VEL
LIN {X 0,Y 156.57,Z 619.222,A -85,B 0,C 180,E1 -23959.5,E2 -23959.5} C_VEL
LIN {X 0,Y 153.798,Z 618.565,A -85,B 0,C 180,E1 -23964.285,E2 -23964.285} C_VEL
LIN {X 0,Y 152.076,Z 616.882,A -85,B 0,C 180,E1 -23968.589,E2 -23968.589} C_VEL
LIN {X 0,Y 150.998,Z 613.352,A -85,B 0,C 180,E1 -23973.955,E2 -23973.955} C_VEL
LIN {X 0,Y 150.854,Z 608.555,A -85,B 0,C 180,E1 -23979.021,E2 -23979.021} C_VEL
LIN {X 0,Y 151.621,Z 602.05,A -85,B 0,C 180,E1 -23984.051,E2 -23984.051} C_VEL
LIN {X 0,Y 152.921,Z 595.281,A -85,B 0,C 180,E1 -23988.131,E2 -23988.131} C_VEL
LIN {X 0,Y 154.684,Z 586.973,A -85,B 0,C 180,E1 -23992.133,E2 -23992.133} C_VEL
LIN {X 0,Y 156.909,Z 576.981,A -85,B 0,C 180,E1 -23995.959,E2 -23995.959} C_VEL
LIN {X 0,Y 159.145,Z 566.997,A -85,B 0,C 180,E1 -23999.016,E2 -23999.016} C_VEL
LIN {X 0,Y 159.872,Z 563.297,A -85,B 0,C 180,E1 -23999.996,E2 -23999.996} C_VEL
LIN {X 0,Y 158.202,Z 555.645,A -85,B 0,C 180,E1 -24002.195,E2 -24002.195} C_VEL
LIN {X 0,Y 155.356,Z 545.299,A -85,B 0,C 180,E1 -24004.904,E2 -24004.904} C_VEL
LIN {X 0,Y 151.688,Z 534.098,A -85,B 0,C 180,E1 -24007.526,E2 -24007.526} C_VEL
LIN {X 0,Y 150.317,Z 529.761,A -85,B 0,C 180,E1 -24008.508,E2 -24008.508} C_VEL
LIN {X 0,Y 150.352,Z 529.759,A -85,B 0,C 180,E1 -24013.712,E2 -24013.712} C_VEL
LIN {X 0,Y 150.614,Z 529.726,A -85,B 0,C 180,E1 -24019.242,E2 -24019.242} C_VEL
LIN {X 0,Y 150.705,Z 529.712,A -85,B 0,C 180,E1 -24021.957,E2 -24021.957} C_VEL
LIN {X 0,Y 151.216,Z 529.648,A -85,B 0,C 180,E1 -24030,E2 -24030} C_VEL
LIN {X 0,Y 150.687,Z 529.709,A -85,B 0,C 180,E1 -24038.043,E2 -24038.043} C_VEL
LIN {X 0,Y 150.578,Z 529.729,A -85,B 0,C 180,E1 -24041.431,E2 -24041.431} C_VEL
LIN {X 0,Y 150.352,Z 529.752,A -85,B 0,C 180,E1 -24046.287,E2 -24046.287} C_VEL
LIN {X 0,Y 150.352,Z 529.756,A -85,B 0,C 180,E1 -24050.79,E2 -24050.79} C_VEL
LIN {X 0,Y 150.241,Z 529.767,A -85,B 0,C 180,E1 -24057.277,E2 -24057.277} C_VEL
LIN {X 0,Y 150.211,Z 529.772,A -85,B 0,C 180,E1 -24062.627,E2 -24062.627} C_VEL
LIN {X 0,Y 150.171,Z 529.779,A -85,B 0,C 180,E1 -24067.474,E2 -24067.474} C_VEL
LIN {X 0,Y 150.136,Z 529.779,A -85,B 0,C 180,E1 -24071.497,E2 -24071.497} C_VEL
LIN {X 0,Y 150.128,Z 529.784,A -85,B 0,C 180,E1 -24075.395,E2 -24075.395} C_VEL
LIN {X 0,Y 150.143,Z 529.782,A -85,B 0,C 180,E1 -24079.055,E2 -24079.055} C_VEL
LIN {X 0,Y 150.181,Z 529.773,A -85,B 0,C 180,E1 -24082.707,E2 -24082.707} C_VEL
LIN {X 0,Y 150.217,Z 529.772,A -85,B 0,C 180,E1 -24087.367,E2 -24087.367} C_VEL
LIN {X 0,Y 150.243,Z 529.768,A -85,B 0,C 180,E1 -24092.72,E2 -24092.72} C_VEL
LIN {X 0,Y 150.351,Z 529.752,A -85,B 0,C 180,E1 -24099.208,E2 -24099.208} C_VEL
LIN {X 0,Y 150.363,Z 529.754,A -85,B 0,C 180,E1 -24103.713,E2 -24103.713} C_VEL
LIN {X 0,Y 150.612,Z 529.723,A -85,B 0,C 180,E1 -24109.242,E2 -24109.242} C_VEL
LIN {X 0,Y 150.702,Z 529.712,A -85,B 0,C 180,E1 -24111.957,E2 -24111.957} C_VEL
LIN {X 0,Y 151.214,Z 529.648,A -85,B 0,C 180,E1 -24119.999,E2 -24119.999} C_VEL
LIN {X 0,Y 150.699,Z 529.712,A -85,B 0,C 180,E1 -24128.042,E2 -24128.042} C_VEL
LIN {X 0,Y 150.575,Z 529.725,A -85,B 0,C 180,E1 -24131.431,E2 -24131.431} C_VEL
LIN {X 0,Y 150.349,Z 529.756,A -85,B 0,C 180,E1 -24136.287,E2 -24136.287} C_VEL
LIN {X 0,Y 150.349,Z 529.752,A -85,B 0,C 180,E1 -24140.789,E2 -24140.789} C_VEL
LIN {X 0,Y 150.238,Z 529.769,A -85,B 0,C 180,E1 -24147.277,E2 -24147.277} C_VEL
LIN {X 0,Y 150.342,Z 529.901,A -85,B 0,C 180,E1 -24152.46,E2 -24152.46} C_VEL
LIN {X 0,Y 151.385,Z 535.316,A -85,B 0,C 180,E1 -24157.887,E2 -24157.887} C_VEL
LIN {X 0,Y 152.628,Z 541.409,A -85,B 0,C 180,E1 -24163.685,E2 -24163.685} C_VEL
LIN {X 0,Y 153.892,Z 547.04,A -85,B 0,C 180,E1 -24168.779,E2 -24168.779} C_VEL
LIN {X 0,Y 153.67,Z 549.664,A -85,B 0,C 180,E1 -24171.03,E2 -24171.03} C_VEL
LIN {X 0,Y 152.76,Z 552.498,A -85,B 0,C 180,E1 -24173.434,E2 -24173.434} C_VEL
LIN {X 0,Y 153.399,Z 567.858,A -85,B 0,C 180,E1 -24175.131,E2 -24175.131} C_VEL
LIN {X 0,Y 153.742,Z 581.021,A -85,B 0,C 180,E1 -24177.123,E2 -24177.123} C_VEL
LIN {X 0,Y 153.713,Z 593.134,A -85,B 0,C 180,E1 -24179.426,E2 -24179.426} C_VEL
LIN {X 0,Y 153.527,Z 604.238,A -85,B 0,C 180,E1 -24182.025,E2 -24182.025} C_VEL
LIN {X 0,Y 153.248,Z 615.467,A -85,B 0,C 180,E1 -24185.262,E2 -24185.262} C_VEL
LIN {X 0,Y 152.857,Z 624.504,A -85,B 0,C 180,E1 -24188.419,E2 -24188.419} C_VEL
LIN {X 0,Y 151.884,Z 630.933,A -85,B 0,C 180,E1 -24191.101,E2 -24191.101} C_VEL
LIN {X 0,Y 150.436,Z 638.769,A -85,B 0,C 180,E1 -24195.111,E2 -24195.111} C_VEL
LIN {X 0,Y 149.989,Z 645.125,A -85,B 0,C 180,E1 -24199.198,E2 -24199.198} C_VEL
LIN {X 0,Y 150.13,Z 650.08,A -85,B 0,C 180,E1 -24203.279,E2 -24203.279} C_VEL
LIN {X 0,Y 150.756,Z 653.797,A -85,B 0,C 180,E1 -24207.328,E2 -24207.328} C_VEL
LIN {X 0,Y 151.249,Z 655.579,A -85,B 0,C 180,E1 -24210,E2 -24210} C_VEL
LIN {X 0,Y 150.473,Z 656.625,A -85,B 0,C 180,E1 -24212.677,E2 -24212.677} C_VEL
LIN {X 0,Y 149.291,Z 657.505,A -85,B 0,C 180,E1 -24218.119,E2 -24218.119} C_VEL
LIN {X 0,Y 149.348,Z 656.911,A -85,B 0,C 180,E1 -24223.609,E2 -24223.609} C_VEL
LIN {X 0,Y 150.917,Z 654.937,A -85,B 0,C 180,E1 -24229.025,E2 -24229.025} C_VEL
LIN {X 0,Y 154.056,Z 651.599,A -85,B 0,C 180,E1 -24234.242,E2 -24234.242} C_VEL
LIN {X 0,Y 158.851,Z 646.836,A -85,B 0,C 180,E1 -24239.123,E2 -24239.123} C_VEL
LIN {X 0,Y 163.044,Z 642.226,A -85,B 0,C 180,E1 -24242.603,E2 -24242.603} C_VEL
LIN {X 0,Y 169.106,Z 634.568,A -85,B 0,C 180,E1 -24247.058,E2 -24247.058} C_VEL
LIN {X 0,Y 173.858,Z 627.68,A -85,B 0,C 180,E1 -24250.3,E2 -24250.3} C_VEL
LIN {X 0,Y 179.154,Z 618.377,A -85,B 0,C 180,E1 -24254.133,E2 -24254.133} C_VEL
LIN {X 0,Y 183.218,Z 609.545,A -85,B 0,C 180,E1 -24257.507,E2 -24257.507} C_VEL
LIN {X 0,Y 185.958,Z 602.851,A -85,B 0,C 180,E1 -24260.023,E2 -24260.023} C_VEL
LIN {X 0,Y 186.428,Z 601.003,A -85,B 0,C 180,E1 -24260.844,E2 -24260.844} C_VEL
LIN {X 0,Y 186.562,Z 597.343,A -85,B 0,C 180,E1 -24263.127,E2 -24263.127} C_VEL
LIN {X 0,Y 186.048,Z 595.626,A -85,B 0,C 180,E1 -24264.857,E2 -24264.857} C_VEL
LIN {X 0,Y 184.953,Z 594.757,A -85,B 0,C 180,E1 -24266.645,E2 -24266.645} C_VEL
LIN {X 0,Y 182.021,Z 593.793,A -85,B 0,C 180,E1 -24271.588,E2 -24271.588} C_VEL
LIN {X 0,Y 181.868,Z 593.241,A -85,B 0,C 180,E1 -24272.845,E2 -24272.845} C_VEL
LIN {X 0,Y 182.069,Z 592.089,A -85,B 0,C 180,E1 -24274.875,E2 -24274.875} C_VEL
LIN {X 0,Y 182.51,Z 591.064,A -85,B 0,C 180,E1 -24277.546,E2 -24277.546} C_VEL
LIN {X 0,Y 182.873,Z 590.641,A -85,B 0,C 180,E1 -24279.765,E2 -24279.765} C_VEL
LIN {X 0,Y 183.386,Z 590.88,A -85,B 0,C 180,E1 -24283.356,E2 -24283.356} C_VEL
LIN {X 0,Y 183.558,Z 591.177,A -85,B 0,C 180,E1 -24284.454,E2 -24284.454} C_VEL
LIN {X 0,Y 183.324,Z 592.56,A -85,B 0,C 180,E1 -24286.702,E2 -24286.702} C_VEL
LIN {X 0,Y 182.348,Z 596.352,A -85,B 0,C 180,E1 -24291.132,E2 -24291.132} C_VEL
LIN {X 0,Y 181.113,Z 599.731,A -85,B 0,C 180,E1 -24294.433,E2 -24294.433} C_VEL
LIN {X 0,Y 179.746,Z 602.349,A -85,B 0,C 180,E1 -24296.638,E2 -24296.638} C_VEL
LIN {X 0,Y 172.908,Z 608.66,A -85,B 0,C 180,E1 -24300.001,E2 -24300.001} C_VEL
LIN {X 0,Y 166.651,Z 613.506,A -85,B 0,C 180,E1 -24303.627,E2 -24303.627} C_VEL
LIN {X 0,Y 160.963,Z 617.006,A -85,B 0,C 180,E1 -24307.527,E2 -24307.527} C_VEL
LIN {X 0,Y 157.295,Z 618.788,A -85,B 0,C 180,E1 -24310.586,E2 -24310.586} C_VEL
LIN {X 0,Y 152.83,Z 620.161,A -85,B 0,C 180,E1 -24315.047,E2 -24315.047} C_VEL
LIN {X 0,Y 149.26,Z 620.323,A -85,B 0,C 180,E1 -24319.657,E2 -24319.657} C_VEL
LIN {X 0,Y 146.608,Z 619.313,A -85,B 0,C 180,E1 -24324.381,E2 -24324.381} C_VEL
LIN {X 0,Y 144.812,Z 617.201,A -85,B 0,C 180,E1 -24329.122,E2 -24329.122} C_VEL
LIN {X 0,Y 143.939,Z 613.951,A -85,B 0,C 180,E1 -24333.895,E2 -24333.895} C_VEL
LIN {X 0,Y 143.817,Z 608.634,A -85,B 0,C 180,E1 -24339.442,E2 -24339.442} C_VEL
LIN {X 0,Y 144.463,Z 603.032,A -85,B 0,C 180,E1 -24343.887,E2 -24343.887} C_VEL
LIN {X 0,Y 145.703,Z 596.606,A -85,B 0,C 180,E1 -24347.969,E2 -24347.969} C_VEL
LIN {X 0,Y 147.377,Z 588.878,A -85,B 0,C 180,E1 -24351.954,E2 -24351.954} C_VEL
LIN {X 0,Y 149.395,Z 579.991,A -85,B 0,C 180,E1 -24355.631,E2 -24355.631} C_VEL
LIN {X 0,Y 151.724,Z 569.981,A -85,B 0,C 180,E1 -24358.957,E2 -24358.957} C_VEL
LIN {X 0,Y 152.898,Z 564.658,A -85,B 0,C 180,E1 -24360.462,E2 -24360.462} C_VEL
LIN {X 0,Y 151.655,Z 558.322,A -85,B 0,C 180,E1 -24362.391,E2 -24362.391} C_VEL
LIN {X 0,Y 148.913,Z 548.167,A -85,B 0,C 180,E1 -24365.237,E2 -24365.237} C_VEL
LIN {X 0,Y 145.628,Z 537.816,A -85,B 0,C 180,E1 -24367.823,E2 -24367.823} C_VEL
LIN {X 0,Y 143.321,Z 530.634,A -85,B 0,C 180,E1 -24369.497,E2 -24369.497} C_VEL
LIN {X 0,Y 143.355,Z 530.63,A -85,B 0,C 180,E1 -24375.81,E2 -24375.81} C_VEL
LIN {X 0,Y 143.54,Z 530.606,A -85,B 0,C 180,E1 -24378.705,E2 -24378.705} C_VEL
LIN {X 0,Y 143.627,Z 530.595,A -85,B 0,C 180,E1 -24381.558,E2 -24381.558} C_VEL
LIN {X 0,Y 144.175,Z 530.525,A -85,B 0,C 180,E1 -24390,E2 -24390} C_VEL
LIN {X 0,Y 143.612,Z 530.59,A -85,B 0,C 180,E1 -24398.442,E2 -24398.442} C_VEL
LIN {X 0,Y 143.504,Z 530.609,A -85,B 0,C 180,E1 -24401.621,E2 -24401.621} C_VEL
LIN {X 0,Y 143.296,Z 530.63,A -85,B 0,C 180,E1 -24407.114,E2 -24407.114} C_VEL
LIN {X 0,Y 143.278,Z 530.639,A -85,B 0,C 180,E1 -24411.251,E2 -24411.251} C_VEL
LIN {X 0,Y 143.185,Z 530.647,A -85,B 0,C 180,E1 -24417.93,E2 -24417.93} C_VEL
LIN {X 0,Y 143.14,Z 530.649,A -85,B 0,C 180,E1 -24423.416,E2 -24423.416} C_VEL
LIN {X 0,Y 143.055,Z 530.664,A -85,B 0,C 180,E1 -24429.692,E2 -24429.692} C_VEL
LIN {X 0,Y 143.035,Z 530.663,A -85,B 0,C 180,E1 -24433.463,E2 -24433.463} C_VEL
LIN {X 0,Y 143.041,Z 530.667,A -85,B 0,C 180,E1 -24437.475,E2 -24437.475} C_VEL
LIN {X 0,Y 143.077,Z 530.657,A -85,B 0,C 180,E1 -24441.806,E2 -24441.806} C_VEL
LIN {X 0,Y 143.184,Z 530.648,A -85,B 0,C 180,E1 -24447.321,E2 -24447.321} C_VEL
LIN {X 0,Y 143.19,Z 530.646,A -85,B 0,C 180,E1 -24452.064,E2 -24452.064} C_VEL
LIN {X 0,Y 143.277,Z 530.632,A -85,B 0,C 180,E1 -24458.746,E2 -24458.746} C_VEL
LIN {X 0,Y 143.303,Z 530.635,A -85,B 0,C 180,E1 -24462.886,E2 -24462.886} C_VEL
LIN {X 0,Y 143.538,Z 530.601,A -85,B 0,C 180,E1 -24468.705,E2 -24468.705} C_VEL
LIN {X 0,Y 143.624,Z 530.594,A -85,B 0,C 180,E1 -24471.558,E2 -24471.558} C_VEL
LIN {X 0,Y 144.173,Z 530.525,A -85,B 0,C 180,E1 -24479.999,E2 -24479.999} C_VEL
LIN {X 0,Y 143.621,Z 530.595,A -85,B 0,C 180,E1 -24488.441,E2 -24488.441} C_VEL
LIN {X 0,Y 143.502,Z 530.605,A -85,B 0,C 180,E1 -24491.621,E2 -24491.621} C_VEL
LIN {X 0,Y 143.292,Z 530.636,A -85,B 0,C 180,E1 -24497.114,E2 -24497.114} C_VEL
LIN {X 0,Y 143.274,Z 530.632,A -85,B 0,C 180,E1 -24501.251,E2 -24501.251} C_VEL
LIN {X 0,Y 143.183,Z 530.647,A -85,B 0,C 180,E1 -24507.931,E2 -24507.931} C_VEL
LIN {X 0,Y 143.298,Z 530.736,A -85,B 0,C 180,E1 -24512.025,E2 -24512.025} C_VEL
LIN {X 0,Y 144.288,Z 535.824,A -85,B 0,C 180,E1 -24517.387,E2 -24517.387} C_VEL
LIN {X 0,Y 145.531,Z 542.014,A -85,B 0,C 180,E1 -24523.583,E2 -24523.583} C_VEL
LIN {X 0,Y 146.803,Z 547.82,A -85,B 0,C 180,E1 -24529.064,E2 -24529.064} C_VEL
LIN {X 0,Y 146.378,Z 550.394,A -85,B 0,C 180,E1 -24531.379,E2 -24531.379} C_VEL
LIN {X 0,Y 146,Z 551.489,A -85,B 0,C 180,E1 -24532.358,E2 -24532.358} C_VEL
LIN {X 0,Y 146.581,Z 567.734,A -85,B 0,C 180,E1 -24534.292,E2 -24534.292} C_VEL
LIN {X 0,Y 146.847,Z 582.032,A -85,B 0,C 180,E1 -24536.607,E2 -24536.607} C_VEL
LIN {X 0,Y 146.732,Z 594.273,A -85,B 0,C 180,E1 -24539.134,E2 -24539.134} C_VEL
LIN {X 0,Y 146.468,Z 605.86,A -85,B 0,C 180,E1 -24542.106,E2 -24542.106} C_VEL
LIN {X 0,Y 146.142,Z 616.644,A -85,B 0,C 180,E1 -24545.486,E2 -24545.486} C_VEL
LIN {X 0,Y 145.7,Z 625.29,A -85,B 0,C 180,E1 -24548.791,E2 -24548.791} C_VEL
LIN {X 0,Y 144.275,Z 632.729,A -85,B 0,C 180,E1 -24552.275,E2 -24552.275} C_VEL
LIN {X 0,Y 143.265,Z 640.015,A -85,B 0,C 180,E1 -24556.526,E2 -24556.526} C_VEL
LIN {X 0,Y 142.998,Z 645.05,A -85,B 0,C 180,E1 -24560.17,E2 -24560.17} C_VEL
LIN {X 0,Y 143.261,Z 649.669,A -85,B 0,C 180,E1 -24564.37,E2 -24564.37} C_VEL
LIN {X 0,Y 143.734,Z 652.138,A -85,B 0,C 180,E1 -24567.198,E2 -24567.198} C_VEL
LIN {X 0,Y 144.265,Z 654.082,A -85,B 0,C 180,E1 -24570,E2 -24570} C_VEL
LIN {X 0,Y 143.455,Z 655.205,A -85,B 0,C 180,E1 -24572.808,E2 -24572.808} C_VEL
LIN {X 0,Y 142.259,Z 656.227,A -85,B 0,C 180,E1 -24578.524,E2 -24578.524} C_VEL
LIN {X 0,Y 142.429,Z 655.838,A -85,B 0,C 180,E1 -24584.284,E2 -24584.284} C_VEL
LIN {X 0,Y 144.166,Z 654.077,A -85,B 0,C 180,E1 -24589.953,E2 -24589.953} C_VEL
LIN {X 0,Y 147.578,Z 650.956,A -85,B 0,C 180,E1 -24595.379,E2 -24595.379} C_VEL
LIN {X 0,Y 152.648,Z 646.447,A -85,B 0,C 180,E1 -24600.428,E2 -24600.428} C_VEL
LIN {X 0,Y 157.03,Z 642.041,A -85,B 0,C 180,E1 -24604.018,E2 -24604.018} C_VEL
LIN {X 0,Y 163.446,Z 634.788,A -85,B 0,C 180,E1 -24608.572,E2 -24608.572} C_VEL
LIN {X 0,Y 168.44,Z 628.208,A -85,B 0,C 180,E1 -24611.882,E2 -24611.882} C_VEL
LIN {X 0,Y 174.082,Z 619.355,A -85,B 0,C 180,E1 -24615.775,E2 -24615.775} C_VEL
LIN {X 0,Y 179.138,Z 609.698,A -85,B 0,C 180,E1 -24619.727,E2 -24619.727} C_VEL
LIN {X 0,Y 181.13,Z 605.152,A -85,B 0,C 180,E1 -24621.625,E2 -24621.625} C_VEL
LIN {X 0,Y 181.569,Z 600.946,A -85,B 0,C 180,E1 -24624.507,E2 -24624.507} C_VEL
LIN {X 0,Y 181.935,Z 596.555,A -85,B 0,C 180,E1 -24628.195,E2 -24628.195} C_VEL
LIN {X 0,Y 181.868,Z 593.241,A -85,B 0,C 180,E1 -24632.845,E2 -24632.845} C_VEL
LIN {X 0,Y 181.57,Z 592.78,A -85,B 0,C 180,E1 -24634.7,E2 -24634.7} C_VEL
LIN {X 0,Y 180.776,Z 593.194,A -85,B 0,C 180,E1 -24636.561,E2 -24636.561} C_VEL
LIN {X 0,Y 178.395,Z 595.655,A -85,B 0,C 180,E1 -24641.589,E2 -24641.589} C_VEL
LIN {X 0,Y 178.33,Z 595.956,A -85,B 0,C 180,E1 -24642.881,E2 -24642.881} C_VEL
LIN {X 0,Y 178.49,Z 596.078,A -85,B 0,C 180,E1 -24644.001,E2 -24644.001} C_VEL
LIN {X 0,Y 178.154,Z 597.271,A -85,B 0,C 180,E1 -24646.309,E2 -24646.309} C_VEL
LIN {X 0,Y 176.766,Z 600.731,A -85,B 0,C 180,E1 -24650.85,E2 -24650.85} C_VEL
LIN {X 0,Y 175.108,Z 603.859,A -85,B 0,C 180,E1 -24654.242,E2 -24654.242} C_VEL
LIN {X 0,Y 174.329,Z 605.103,A -85,B 0,C 180,E1 -24655.376,E2 -24655.376} C_VEL
LIN {X 0,Y 167.194,Z 611.057,A -85,B 0,C 180,E1 -24658.795,E2 -24658.795} C_VEL
LIN {X 0,Y 160.612,Z 615.566,A -85,B 0,C 180,E1 -24662.509,E2 -24662.509} C_VEL
LIN {X 0,Y 155.454,Z 618.415,A -85,B 0,C 180,E1 -24665.944,E2 -24665.944} C_VEL
LIN {X 0,Y 149.55,Z 620.783,A -85,B 0,C 180,E1 -24670.836,E2 -24670.836} C_VEL
LIN {X 0,Y 145.513,Z 621.566,A -85,B 0,C 180,E1 -24674.989,E2 -24674.989} C_VEL
LIN {X 0,Y 141.596,Z 621.191,A -85,B 0,C 180,E1 -24680.332,E2 -24680.332} C_VEL
LIN {X 0,Y 139.295,Z 619.884,A -85,B 0,C 180,E1 -24684.744,E2 -24684.744} C_VEL
LIN {X 0,Y 137.327,Z 616.71,A -85,B 0,C 180,E1 -24690.783,E2 -24690.783} C_VEL
LIN {X 0,Y 136.674,Z 612.369,A -85,B 0,C 180,E1 -24696.282,E2 -24696.282} C_VEL
LIN {X 0,Y 136.983,Z 606.422,A -85,B 0,C 180,E1 -24701.835,E2 -24701.835} C_VEL
LIN {X 0,Y 138.029,Z 600.137,A -85,B 0,C 180,E1 -24706.391,E2 -24706.391} C_VEL
LIN {X 0,Y 139.806,Z 591.744,A -85,B 0,C 180,E1 -24711.187,E2 -24711.187} C_VEL
LIN {X 0,Y 141.971,Z 582.512,A -85,B 0,C 180,E1 -24715.385,E2 -24715.385} C_VEL
LIN {X 0,Y 144.518,Z 571.869,A -85,B 0,C 180,E1 -24719.198,E2 -24719.198} C_VEL
LIN {X 0,Y 145.972,Z 565.135,A -85,B 0,C 180,E1 -24721.218,E2 -24721.218} C_VEL
LIN {X 0,Y 143.666,Z 555.422,A -85,B 0,C 180,E1 -24724.268,E2 -24724.268} C_VEL
LIN {X 0,Y 140.874,Z 545.631,A -85,B 0,C 180,E1 -24727.033,E2 -24727.033} C_VEL
LIN {X 0,Y 136.844,Z 533.544,A -85,B 0,C 180,E1 -24730.108,E2 -24730.108} C_VEL
LIN {X 0,Y 136.227,Z 531.517,A -85,B 0,C 180,E1 -24730.602,E2 -24730.602} C_VEL
LIN {X 0,Y 136.446,Z 531.49,A -85,B 0,C 180,E1 -24738.144,E2 -24738.144} C_VEL
LIN {X 0,Y 136.553,Z 531.478,A -85,B 0,C 180,E1 -24741.117,E2 -24741.117} C_VEL
LIN {X 0,Y 137.133,Z 531.403,A -85,B 0,C 180,E1 -24750,E2 -24750} C_VEL
LIN {X 0,Y 136.541,Z 531.471,A -85,B 0,C 180,E1 -24758.883,E2 -24758.883} C_VEL
LIN {X 0,Y 136.424,Z 531.491,A -85,B 0,C 180,E1 -24761.891,E2 -24761.891} C_VEL
LIN {X 0,Y 136.239,Z 531.509,A -85,B 0,C 180,E1 -24768.03,E2 -24768.03} C_VEL
LIN {X 0,Y 136.198,Z 531.519,A -85,B 0,C 180,E1 -24771.745,E2 -24771.745} C_VEL
LIN {X 0,Y 136.095,Z 531.531,A -85,B 0,C 180,E1 -24778.609,E2 -24778.609} C_VEL
LIN {X 0,Y 136.042,Z 531.532,A -85,B 0,C 180,E1 -24784.629,E2 -24784.629} C_VEL
LIN {X 0,Y 136.027,Z 531.542,A -85,B 0,C 180,E1 -24789.194,E2 -24789.194} C_VEL
LIN {X 0,Y 135.98,Z 531.542,A -85,B 0,C 180,E1 -24793.648,E2 -24793.648} C_VEL
LIN {X 0,Y 135.986,Z 531.545,A -85,B 0,C 180,E1 -24797.787,E2 -24797.787} C_VEL
LIN {X 0,Y 136.026,Z 531.535,A -85,B 0,C 180,E1 -24801.683,E2 -24801.683} C_VEL
LIN {X 0,Y 136.087,Z 531.533,A -85,B 0,C 180,E1 -24805.72,E2 -24805.72} C_VEL
LIN {X 0,Y 136.146,Z 531.523,A -85,B 0,C 180,E1 -24812.315,E2 -24812.315} C_VEL
LIN {X 0,Y 136.244,Z 531.508,A -85,B 0,C 180,E1 -24818.832,E2 -24818.832} C_VEL
LIN {X 0,Y 136.27,Z 531.509,A -85,B 0,C 180,E1 -24825.055,E2 -24825.055} C_VEL
LIN {X 0,Y 136.433,Z 531.485,A -85,B 0,C 180,E1 -24828.164,E2 -24828.164} C_VEL
LIN {X 0,Y 136.55,Z 531.477,A -85,B 0,C 180,E1 -24831.117,E2 -24831.117} C_VEL
LIN {X 0,Y 137.13,Z 531.403,A -85,B 0,C 180,E1 -24839.999,E2 -24839.999} C_VEL
LIN {X 0,Y 136.547,Z 531.477,A -85,B 0,C 180,E1 -24848.882,E2 -24848.882} C_VEL
LIN {X 0,Y 136.418,Z 531.487,A -85,B 0,C 180,E1 -24851.892,E2 -24851.892} C_VEL
LIN {X 0,Y 136.236,Z 531.514,A -85,B 0,C 180,E1 -24858.03,E2 -24858.03} C_VEL
LIN {X 0,Y 136.195,Z 531.513,A -85,B 0,C 180,E1 -24861.745,E2 -24861.745} C_VEL
LIN {X 0,Y 136.112,Z 531.527,A -85,B 0,C 180,E1 -24868.625,E2 -24868.625} C_VEL
LIN {X 0,Y 136.235,Z 531.654,A -85,B 0,C 180,E1 -24871.704,E2 -24871.704} C_VEL
LIN {X 0,Y 137.008,Z 535.647,A -85,B 0,C 180,E1 -24876.148,E2 -24876.148} C_VEL
LIN {X 0,Y 138.033,Z 540.626,A -85,B 0,C 180,E1 -24881.444,E2 -24881.444} C_VEL
LIN {X 0,Y 139.24,Z 546.191,A -85,B 0,C 180,E1 -24887.043,E2 -24887.043} C_VEL
LIN {X 0,Y 139.732,Z 548.369,A -85,B 0,C 180,E1 -24889.167,E2 -24889.167} C_VEL
LIN {X 0,Y 139.228,Z 550.723,A -85,B 0,C 180,E1 -24891.285,E2 -24891.285} C_VEL
LIN {X 0,Y 139.719,Z 565.316,A -85,B 0,C 180,E1 -24893.033,E2 -24893.033} C_VEL
LIN {X 0,Y 139.919,Z 578.787,A -85,B 0,C 180,E1 -24895.253,E2 -24895.253} C_VEL
LIN {X 0,Y 139.823,Z 591.41,A -85,B 0,C 180,E1 -24897.898,E2 -24897.898} C_VEL
LIN {X 0,Y 139.518,Z 603.269,A -85,B 0,C 180,E1 -24900.998,E2 -24900.998} C_VEL
